LIN {X 0,Y 411.222,Z 293.884,A -85,B 0,C 180,E1 -10421.051,E2 -10421.051} C_VEL
LIN {X 0,Y 411.251,Z 293.88,A -85,B 0,C 180,E1 -10424.131,E2 -10424.131} C_VEL
LIN {X 0,Y 411.3,Z 293.873,A -85,B 0,C 180,E1 -10427.165,E2 -10427.165} C_VEL
LIN {X 0,Y 411.29,Z 293.877,A -85,B 0,C 180,E1 -10430.161,E2 -10430.161} C_VEL
LIN {X 0,Y 411.391,Z 293.865,A -85,B 0,C 180,E1 -10433.132,E2 -10433.132} C_VEL
LIN {X 0,Y 411.304,Z 293.877,A -85,B 0,C 180,E1 -10435.099,E2 -10435.099} C_VEL
LIN {X 0,Y 411.511,Z 293.85,A -85,B 0,C 180,E1 -10438.042,E2 -10438.042} C_VEL
LIN {X 0,Y 411.632,Z 293.838,A -85,B 0,C 180,E1 -10440,E2 -10440} C_VEL
LIN {X 0,Y 411.464,Z 293.859,A -85,B 0,C 180,E1 -10442.937,E2 -10442.937} C_VEL
LIN {X 0,Y 411.433,Z 293.861,A -85,B 0,C 180,E1 -10445.882,E2 -10445.882} C_VEL
LIN {X 0,Y 411.316,Z 293.875,A -85,B 0,C 180,E1 -10448.846,E2 -10448.846} C_VEL
LIN {X 0,Y 411.281,Z 293.88,A -85,B 0,C 180,E1 -10451.833,E2 -10451.833} C_VEL
LIN {X 0,Y 411.256,Z 293.883,A -85,B 0,C 180,E1 -10454.853,E2 -10454.853} C_VEL
LIN {X 0,Y 411.249,Z 293.883,A -85,B 0,C 180,E1 -10457.915,E2 -10457.915} C_VEL
LIN {X 0,Y 411.193,Z 293.89,A -85,B 0,C 180,E1 -10461.034,E2 -10461.034} C_VEL
LIN {X 0,Y 411.217,Z 293.888,A -85,B 0,C 180,E1 -10464.216,E2 -10464.216} C_VEL
LIN {X 0,Y 411.256,Z 293.886,A -85,B 0,C 180,E1 -10467.478,E2 -10467.478} C_VEL
LIN {X 0,Y 411.187,Z 293.897,A -85,B 0,C 180,E1 -10470.848,E2 -10470.848} C_VEL
LIN {X 0,Y 411.203,Z 293.895,A -85,B 0,C 180,E1 -10474.334,E2 -10474.334} C_VEL
LIN {X 0,Y 411.188,Z 293.897,A -85,B 0,C 180,E1 -10477.974,E2 -10477.974} C_VEL
LIN {X 0,Y 411.158,Z 293.897,A -85,B 0,C 180,E1 -10481.228,E2 -10481.228} C_VEL
LIN {X 0,Y 411.22,Z 294.123,A -85,B 0,C 180,E1 -10483.127,E2 -10483.127} C_VEL
LIN {X 0,Y 411.74,Z 297.377,A -85,B 0,C 180,E1 -10485.799,E2 -10485.799} C_VEL
LIN {X 0,Y 412.024,Z 301.04,A -85,B 0,C 180,E1 -10488.635,E2 -10488.635} C_VEL
LIN {X 0,Y 411.836,Z 305.321,A -85,B 0,C 180,E1 -10491.72,E2 -10491.72} C_VEL
LIN {X 0,Y 411.501,Z 310.164,A -85,B 0,C 180,E1 -10495.063,E2 -10495.063} C_VEL
LIN {X 0,Y 411.137,Z 315.732,A -85,B 0,C 180,E1 -10498.727,E2 -10498.727} C_VEL
LIN {X 0,Y 410.779,Z 321.654,A -85,B 0,C 180,E1 -10502.488,E2 -10502.488} C_VEL
LIN {X 0,Y 410.569,Z 325.761,A -85,B 0,C 180,E1 -10505.017,E2 -10505.017} C_VEL
LIN {X 0,Y 412.96,Z 333.703,A -85,B 0,C 180,E1 -10505.349,E2 -10505.349} C_VEL
LIN {X 0,Y 417.044,Z 348.163,A -85,B 0,C 180,E1 -10506.057,E2 -10506.057} C_VEL
LIN {X 0,Y 420.257,Z 362.682,A -85,B 0,C 180,E1 -10506.892,E2 -10506.892} C_VEL
LIN {X 0,Y 419.468,Z 375.628,A -85,B 0,C 180,E1 -10507.594,E2 -10507.594} C_VEL
LIN {X 0,Y 418.211,Z 389.915,A -85,B 0,C 180,E1 -10508.561,E2 -10508.561} C_VEL
LIN {X 0,Y 416.924,Z 402.918,A -85,B 0,C 180,E1 -10509.655,E2 -10509.655} C_VEL
LIN {X 0,Y 415.653,Z 414.924,A -85,B 0,C 180,E1 -10510.877,E2 -10510.877} C_VEL
LIN {X 0,Y 414.497,Z 426.042,A -85,B 0,C 180,E1 -10512.23,E2 -10512.23} C_VEL
LIN {X 0,Y 413.333,Z 436.268,A -85,B 0,C 180,E1 -10513.707,E2 -10513.707} C_VEL
LIN {X 0,Y 412.281,Z 446.263,A -85,B 0,C 180,E1 -10515.437,E2 -10515.437} C_VEL
LIN {X 0,Y 411.345,Z 455.643,A -85,B 0,C 180,E1 -10517.418,E2 -10517.418} C_VEL
LIN {X 0,Y 410.772,Z 462.357,A -85,B 0,C 180,E1 -10519.152,E2 -10519.152} C_VEL
LIN {X 0,Y 410.337,Z 468.557,A -85,B 0,C 180,E1 -10521.132,E2 -10521.132} C_VEL
LIN {X 0,Y 410.082,Z 473.352,A -85,B 0,C 180,E1 -10523.11,E2 -10523.11} C_VEL
LIN {X 0,Y 409.968,Z 476.864,A -85,B 0,C 180,E1 -10525.083,E2 -10525.083} C_VEL
LIN {X 0,Y 409.871,Z 479.174,A -85,B 0,C 180,E1 -10527.051,E2 -10527.051} C_VEL
LIN {X 0,Y 409.915,Z 480.337,A -85,B 0,C 180,E1 -10529.017,E2 -10529.017} C_VEL
LIN {X 0,Y 409.915,Z 480.336,A -85,B 0,C 180,E1 -10530.982,E2 -10530.982} C_VEL
LIN {X 0,Y 409.871,Z 479.168,A -85,B 0,C 180,E1 -10532.948,E2 -10532.948} C_VEL
LIN {X 0,Y 409.973,Z 476.855,A -85,B 0,C 180,E1 -10534.917,E2 -10534.917} C_VEL
LIN {X 0,Y 410.155,Z 473.347,A -85,B 0,C 180,E1 -10536.888,E2 -10536.888} C_VEL
LIN {X 0,Y 410.336,Z 468.551,A -85,B 0,C 180,E1 -10538.867,E2 -10538.867} C_VEL
LIN {X 0,Y 410.77,Z 462.34,A -85,B 0,C 180,E1 -10540.847,E2 -10540.847} C_VEL
LIN {X 0,Y 411.351,Z 455.622,A -85,B 0,C 180,E1 -10542.581,E2 -10542.581} C_VEL
LIN {X 0,Y 412.28,Z 446.241,A -85,B 0,C 180,E1 -10544.562,E2 -10544.562} C_VEL
LIN {X 0,Y 413.305,Z 436.241,A -85,B 0,C 180,E1 -10546.294,E2 -10546.294} C_VEL
LIN {X 0,Y 414.63,Z 424.769,A -85,B 0,C 180,E1 -10547.932,E2 -10547.932} C_VEL
LIN {X 0,Y 415.905,Z 412.674,A -85,B 0,C 180,E1 -10549.367,E2 -10549.367} C_VEL
LIN {X 0,Y 417.181,Z 400.249,A -85,B 0,C 180,E1 -10550.589,E2 -10550.589} C_VEL
LIN {X 0,Y 418.477,Z 386.636,A -85,B 0,C 180,E1 -10551.682,E2 -10551.682} C_VEL
LIN {X 0,Y 419.727,Z 372.535,A -85,B 0,C 180,E1 -10552.585,E2 -10552.585} C_VEL
LIN {X 0,Y 420.235,Z 362.738,A -85,B 0,C 180,E1 -10553.101,E2 -10553.101} C_VEL
LIN {X 0,Y 417.1,Z 348.446,A -85,B 0,C 180,E1 -10553.923,E2 -10553.923} C_VEL
LIN {X 0,Y 412.798,Z 333.269,A -85,B 0,C 180,E1 -10554.663,E2 -10554.663} C_VEL
LIN {X 0,Y 410.566,Z 325.765,A -85,B 0,C 180,E1 -10554.987,E2 -10554.987} C_VEL
LIN {X 0,Y 410.775,Z 321.686,A -85,B 0,C 180,E1 -10557.512,E2 -10557.512} C_VEL
LIN {X 0,Y 411.141,Z 315.788,A -85,B 0,C 180,E1 -10561.274,E2 -10561.274} C_VEL
LIN {X 0,Y 411.505,Z 310.225,A -85,B 0,C 180,E1 -10564.937,E2 -10564.937} C_VEL
LIN {X 0,Y 411.833,Z 305.34,A -85,B 0,C 180,E1 -10568.28,E2 -10568.28} C_VEL
LIN {X 0,Y 412.015,Z 300.592,A -85,B 0,C 180,E1 -10571.7,E2 -10571.7} C_VEL
LIN {X 0,Y 411.705,Z 297.085,A -85,B 0,C 180,E1 -10574.417,E2 -10574.417} C_VEL
LIN {X 0,Y 411.217,Z 294.096,A -85,B 0,C 180,E1 -10576.872,E2 -10576.872} C_VEL
LIN {X 0,Y 411.208,Z 293.892,A -85,B 0,C 180,E1 -10580.271,E2 -10580.271} C_VEL
LIN {X 0,Y 411.186,Z 293.896,A -85,B 0,C 180,E1 -10583.447,E2 -10583.447} C_VEL
LIN {X 0,Y 411.2,Z 293.894,A -85,B 0,C 180,E1 -10586.873,E2 -10586.873} C_VEL
LIN {X 0,Y 411.225,Z 293.891,A -85,B 0,C 180,E1 -10590.644,E2 -10590.644} C_VEL
LIN {X 0,Y 411.23,Z 293.888,A -85,B 0,C 180,E1 -10593.619,E2 -10593.619} C_VEL
LIN {X 0,Y 411.195,Z 293.891,A -85,B 0,C 180,E1 -10596.852,E2 -10596.852} C_VEL
LIN {X 0,Y 411.207,Z 293.89,A -85,B 0,C 180,E1 -10600.05,E2 -10600.05} C_VEL
LIN {X 0,Y 411.255,Z 293.883,A -85,B 0,C 180,E1 -10603.131,E2 -10603.131} C_VEL
LIN {X 0,Y 411.297,Z 293.877,A -85,B 0,C 180,E1 -10606.896,E2 -10606.896} C_VEL
LIN {X 0,Y 411.285,Z 293.878,A -85,B 0,C 180,E1 -10610.161,E2 -10610.161} C_VEL
LIN {X 0,Y 411.386,Z 293.865,A -85,B 0,C 180,E1 -10613.132,E2 -10613.132} C_VEL
LIN {X 0,Y 411.301,Z 293.875,A -85,B 0,C 180,E1 -10615.099,E2 -10615.099} C_VEL
LIN {X 0,Y 411.506,Z 293.848,A -85,B 0,C 180,E1 -10618.043,E2 -10618.043} C_VEL
LIN {X 0,Y 411.629,Z 293.838,A -85,B 0,C 180,E1 -10620,E2 -10620} C_VEL
LIN {X 0,Y 411.46,Z 293.859,A -85,B 0,C 180,E1 -10622.937,E2 -10622.937} C_VEL
LIN {X 0,Y 411.389,Z 293.864,A -85,B 0,C 180,E1 -10626.45,E2 -10626.45} C_VEL
LIN {X 0,Y 411.311,Z 293.873,A -85,B 0,C 180,E1 -10628.846,E2 -10628.846} C_VEL
LIN {X 0,Y 411.276,Z 293.877,A -85,B 0,C 180,E1 -10631.833,E2 -10631.833} C_VEL
LIN {X 0,Y 411.251,Z 293.881,A -85,B 0,C 180,E1 -10634.853,E2 -10634.853} C_VEL
LIN {X 0,Y 411.245,Z 293.882,A -85,B 0,C 180,E1 -10637.916,E2 -10637.916} C_VEL
LIN {X 0,Y 411.189,Z 293.89,A -85,B 0,C 180,E1 -10641.035,E2 -10641.035} C_VEL
LIN {X 0,Y 411.22,Z 293.888,A -85,B 0,C 180,E1 -10644.216,E2 -10644.216} C_VEL
LIN {X 0,Y 411.252,Z 293.884,A -85,B 0,C 180,E1 -10647.478,E2 -10647.478} C_VEL
LIN {X 0,Y 411.183,Z 293.89,A -85,B 0,C 180,E1 -10650.848,E2 -10650.848} C_VEL
LIN {X 0,Y 411.199,Z 293.887,A -85,B 0,C 180,E1 -10654.334,E2 -10654.334} C_VEL
LIN {X 0,Y 411.191,Z 293.892,A -85,B 0,C 180,E1 -10657.974,E2 -10657.974} C_VEL
LIN {X 0,Y 411.178,Z 293.893,A -85,B 0,C 180,E1 -10660.505,E2 -10660.505} C_VEL
LIN {X 0,Y 411.168,Z 293.895,A -85,B 0,C 180,E1 -10663.134,E2 -10663.134} C_VEL
LIN {X 0,Y 411.172,Z 293.896,A -85,B 0,C 180,E1 -10664.491,E2 -10664.491} C_VEL
LIN {X 0,Y 411.298,Z 294.707,A -85,B 0,C 180,E1 -10665.863,E2 -10665.863} C_VEL
LIN {X 0,Y 411.549,Z 297.88,A -85,B 0,C 180,E1 -10668.711,E2 -10668.711} C_VEL
LIN {X 0,Y 411.484,Z 300.347,A -85,B 0,C 180,E1 -10670.807,E2 -10670.807} C_VEL
LIN {X 0,Y 411.247,Z 304.858,A -85,B 0,C 180,E1 -10674.477,E2 -10674.477} C_VEL
LIN {X 0,Y 410.983,Z 309.361,A -85,B 0,C 180,E1 -10677.988,E2 -10677.988} C_VEL
LIN {X 0,Y 410.73,Z 313.896,A -85,B 0,C 180,E1 -10681.374,E2 -10681.374} C_VEL
LIN {X 0,Y 410.532,Z 319.007,A -85,B 0,C 180,E1 -10685.077,E2 -10685.077} C_VEL
LIN {X 0,Y 412.277,Z 324.668,A -85,B 0,C 180,E1 -10685.319,E2 -10685.319} C_VEL
LIN {X 0,Y 416.954,Z 339.922,A -85,B 0,C 180,E1 -10686.073,E2 -10686.073} C_VEL
LIN {X 0,Y 420.328,Z 353.637,A -85,B 0,C 180,E1 -10686.87,E2 -10686.87} C_VEL
LIN {X 0,Y 420.411,Z 357.047,A -85,B 0,C 180,E1 -10687.046,E2 -10687.046} C_VEL
LIN {X 0,Y 419.384,Z 371.28,A -85,B 0,C 180,E1 -10687.85,E2 -10687.85} C_VEL
LIN {X 0,Y 418.122,Z 384.886,A -85,B 0,C 180,E1 -10688.816,E2 -10688.816} C_VEL
LIN {X 0,Y 416.783,Z 398.69,A -85,B 0,C 180,E1 -10690.035,E2 -10690.035} C_VEL
LIN {X 0,Y 415.437,Z 411.499,A -85,B 0,C 180,E1 -10691.422,E2 -10691.422} C_VEL
LIN {X 0,Y 414.159,Z 423.349,A -85,B 0,C 180,E1 -10692.98,E2 -10692.98} C_VEL
LIN {X 0,Y 412.951,Z 434.189,A -85,B 0,C 180,E1 -10694.705,E2 -10694.705} C_VEL
LIN {X 0,Y 411.883,Z 443.751,A -85,B 0,C 180,E1 -10696.556,E2 -10696.556} C_VEL
LIN {X 0,Y 411.341,Z 450.645,A -85,B 0,C 180,E1 -10698.17,E2 -10698.17} C_VEL
LIN {X 0,Y 410.673,Z 457.62,A -85,B 0,C 180,E1 -10700.147,E2 -10700.147} C_VEL
LIN {X 0,Y 410.272,Z 463.102,A -85,B 0,C 180,E1 -10702.124,E2 -10702.124} C_VEL
LIN {X 0,Y 410.06,Z 467.242,A -85,B 0,C 180,E1 -10704.098,E2 -10704.098} C_VEL
LIN {X 0,Y 409.919,Z 470.153,A -85,B 0,C 180,E1 -10706.068,E2 -10706.068} C_VEL
LIN {X 0,Y 409.964,Z 471.904,A -85,B 0,C 180,E1 -10708.036,E2 -10708.036} C_VEL
LIN {X 0,Y 409.904,Z 472.517,A -85,B 0,C 180,E1 -10710,E2 -10710} C_VEL
LIN {X 0,Y 409.965,Z 471.952,A -85,B 0,C 180,E1 -10711.965,E2 -10711.965} C_VEL
LIN {X 0,Y 409.918,Z 470.264,A -85,B 0,C 180,E1 -10713.933,E2 -10713.933} C_VEL
LIN {X 0,Y 410.053,Z 467.413,A -85,B 0,C 180,E1 -10715.903,E2 -10715.903} C_VEL
LIN {X 0,Y 410.169,Z 465.034,A -85,B 0,C 180,E1 -10717.121,E2 -10717.121} C_VEL
LIN {X 0,Y 409.551,Z 463.32,A -85,B 0,C 180,E1 -10717.907,E2 -10717.907} C_VEL
LIN {X 0,Y 406.84,Z 460.256,A -85,B 0,C 180,E1 -10719.179,E2 -10719.179} C_VEL
LIN {X 0,Y 404.299,Z 456.695,A -85,B 0,C 180,E1 -10720.439,E2 -10720.439} C_VEL
LIN {X 0,Y 403.951,Z 454.165,A -85,B 0,C 180,E1 -10721.196,E2 -10721.196} C_VEL
LIN {X 0,Y 404.536,Z 448.082,A -85,B 0,C 180,E1 -10722.798,E2 -10722.798} C_VEL
LIN {X 0,Y 405.494,Z 438.803,A -85,B 0,C 180,E1 -10724.812,E2 -10724.812} C_VEL
LIN {X 0,Y 406.669,Z 428.898,A -85,B 0,C 180,E1 -10726.568,E2 -10726.568} C_VEL
LIN {X 0,Y 408.059,Z 417.47,A -85,B 0,C 180,E1 -10728.24,E2 -10728.24} C_VEL
LIN {X 0,Y 409.4,Z 405.552,A -85,B 0,C 180,E1 -10729.688,E2 -10729.688} C_VEL
LIN {X 0,Y 410.75,Z 393.245,A -85,B 0,C 180,E1 -10730.927,E2 -10730.927} C_VEL
LIN {X 0,Y 412.036,Z 379.795,A -85,B 0,C 180,E1 -10732.04,E2 -10732.04} C_VEL
LIN {X 0,Y 413.285,Z 365.857,A -85,B 0,C 180,E1 -10732.958,E2 -10732.958} C_VEL
LIN {X 0,Y 413.862,Z 355.692,A -85,B 0,C 180,E1 -10733.508,E2 -10733.508} C_VEL
LIN {X 0,Y 410.314,Z 341.226,A -85,B 0,C 180,E1 -10734.391,E2 -10734.391} C_VEL
LIN {X 0,Y 405.961,Z 326.76,A -85,B 0,C 180,E1 -10735.144,E2 -10735.144} C_VEL
LIN {X 0,Y 403.515,Z 319.575,A -85,B 0,C 180,E1 -10735.471,E2 -10735.471} C_VEL
LIN {X 0,Y 403.469,Z 319.059,A -85,B 0,C 180,E1 -10735.524,E2 -10735.524} C_VEL
LIN {X 0,Y 403.738,Z 314.147,A -85,B 0,C 180,E1 -10739.17,E2 -10739.17} C_VEL
LIN {X 0,Y 403.985,Z 309.636,A -85,B 0,C 180,E1 -10742.636,E2 -10742.636} C_VEL
LIN {X 0,Y 404.206,Z 306.384,A -85,B 0,C 180,E1 -10745.195,E2 -10745.195} C_VEL
LIN {X 0,Y 404.409,Z 302.079,A -85,B 0,C 180,E1 -10748.728,E2 -10748.728} C_VEL
LIN {X 0,Y 404.552,Z 299.055,A -85,B 0,C 180,E1 -10751.311,E2 -10751.311} C_VEL
LIN {X 0,Y 404.348,Z 296.014,A -85,B 0,C 180,E1 -10754.046,E2 -10754.046} C_VEL
LIN {X 0,Y 404.15,Z 294.772,A -85,B 0,C 180,E1 -10755.477,E2 -10755.477} C_VEL
LIN {X 0,Y 404.118,Z 294.773,A -85,B 0,C 180,E1 -10758.635,E2 -10758.635} C_VEL
LIN {X 0,Y 404.154,Z 294.769,A -85,B 0,C 180,E1 -10761.492,E2 -10761.492} C_VEL
LIN {X 0,Y 404.183,Z 294.768,A -85,B 0,C 180,E1 -10764.984,E2 -10764.984} C_VEL
LIN {X 0,Y 404.14,Z 294.77,A -85,B 0,C 180,E1 -10768.553,E2 -10768.553} C_VEL
LIN {X 0,Y 404.155,Z 294.769,A -85,B 0,C 180,E1 -10770.863,E2 -10770.863} C_VEL
LIN {X 0,Y 404.148,Z 294.77,A -85,B 0,C 180,E1 -10774.231,E2 -10774.231} C_VEL
LIN {X 0,Y 404.165,Z 294.764,A -85,B 0,C 180,E1 -10777.508,E2 -10777.508} C_VEL
LIN {X 0,Y 404.163,Z 294.763,A -85,B 0,C 180,E1 -10780.707,E2 -10780.707} C_VEL
LIN {X 0,Y 404.218,Z 294.756,A -85,B 0,C 180,E1 -10783.848,E2 -10783.848} C_VEL
LIN {X 0,Y 404.28,Z 294.747,A -85,B 0,C 180,E1 -10786.939,E2 -10786.939} C_VEL
LIN {X 0,Y 404.255,Z 294.754,A -85,B 0,C 180,E1 -10789.988,E2 -10789.988} C_VEL
LIN {X 0,Y 404.341,Z 294.743,A -85,B 0,C 180,E1 -10793.011,E2 -10793.011} C_VEL
LIN {X 0,Y 404.274,Z 294.752,A -85,B 0,C 180,E1 -10795.013,E2 -10795.013} C_VEL
LIN {X 0,Y 404.48,Z 294.726,A -85,B 0,C 180,E1 -10798.008,E2 -10798.008} C_VEL
LIN {X 0,Y 404.601,Z 294.713,A -85,B 0,C 180,E1 -10800,E2 -10800} C_VEL
LIN {X 0,Y 404.421,Z 294.736,A -85,B 0,C 180,E1 -10802.988,E2 -10802.988} C_VEL
LIN {X 0,Y 404.381,Z 294.74,A -85,B 0,C 180,E1 -10805.985,E2 -10805.985} C_VEL
LIN {X 0,Y 404.263,Z 294.755,A -85,B 0,C 180,E1 -10809.002,E2 -10809.002} C_VEL
LIN {X 0,Y 404.253,Z 294.757,A -85,B 0,C 180,E1 -10812.041,E2 -10812.041} C_VEL
LIN {X 0,Y 404.202,Z 294.763,A -85,B 0,C 180,E1 -10815.118,E2 -10815.118} C_VEL
LIN {X 0,Y 404.207,Z 294.762,A -85,B 0,C 180,E1 -10818.238,E2 -10818.238} C_VEL
LIN {X 0,Y 404.135,Z 294.772,A -85,B 0,C 180,E1 -10821.419,E2 -10821.419} C_VEL
LIN {X 0,Y 404.171,Z 294.767,A -85,B 0,C 180,E1 -10824.666,E2 -10824.666} C_VEL
LIN {X 0,Y 404.192,Z 294.765,A -85,B 0,C 180,E1 -10828,E2 -10828} C_VEL
LIN {X 0,Y 404.136,Z 294.773,A -85,B 0,C 180,E1 -10831.558,E2 -10831.558} C_VEL
LIN {X 0,Y 404.182,Z 294.771,A -85,B 0,C 180,E1 -10835.016,E2 -10835.016} C_VEL
LIN {X 0,Y 404.146,Z 294.773,A -85,B 0,C 180,E1 -10838.758,E2 -10838.758} C_VEL
LIN {X 0,Y 404.117,Z 294.775,A -85,B 0,C 180,E1 -10841.599,E2 -10841.599} C_VEL
LIN {X 0,Y 404.159,Z 294.854,A -85,B 0,C 180,E1 -10842.701,E2 -10842.701} C_VEL
LIN {X 0,Y 404.687,Z 298.05,A -85,B 0,C 180,E1 -10845.4,E2 -10845.4} C_VEL
LIN {X 0,Y 405.009,Z 301.655,A -85,B 0,C 180,E1 -10848.259,E2 -10848.259} C_VEL
LIN {X 0,Y 404.821,Z 305.87,A -85,B 0,C 180,E1 -10851.373,E2 -10851.373} C_VEL
LIN {X 0,Y 404.471,Z 311.053,A -85,B 0,C 180,E1 -10855.012,E2 -10855.012} C_VEL
LIN {X 0,Y 404.112,Z 316.324,A -85,B 0,C 180,E1 -10858.551,E2 -10858.551} C_VEL
LIN {X 0,Y 403.755,Z 321.601,A -85,B 0,C 180,E1 -10861.967,E2 -10861.967} C_VEL
LIN {X 0,Y 403.516,Z 325.685,A -85,B 0,C 180,E1 -10864.549,E2 -10864.549} C_VEL
LIN {X 0,Y 405.401,Z 331.748,A -85,B 0,C 180,E1 -10864.815,E2 -10864.815} C_VEL
LIN {X 0,Y 409.888,Z 347.21,A -85,B 0,C 180,E1 -10865.58,E2 -10865.58} C_VEL
LIN {X 0,Y 413.149,Z 361.479,A -85,B 0,C 180,E1 -10866.413,E2 -10866.413} C_VEL
LIN {X 0,Y 413.665,Z 364.983,A -85,B 0,C 180,E1 -10866.623,E2 -10866.623} C_VEL
LIN {X 0,Y 412.55,Z 379.541,A -85,B 0,C 180,E1 -10867.462,E2 -10867.462} C_VEL
LIN {X 0,Y 411.285,Z 393.014,A -85,B 0,C 180,E1 -10868.445,E2 -10868.445} C_VEL
LIN {X 0,Y 409.959,Z 405.437,A -85,B 0,C 180,E1 -10869.556,E2 -10869.556} C_VEL
LIN {X 0,Y 408.552,Z 418.07,A -85,B 0,C 180,E1 -10870.923,E2 -10870.923} C_VEL
LIN {X 0,Y 407.269,Z 429.545,A -85,B 0,C 180,E1 -10872.423,E2 -10872.423} C_VEL
LIN {X 0,Y 406.119,Z 439.202,A -85,B 0,C 180,E1 -10873.926,E2 -10873.926} C_VEL
LIN {X 0,Y 405.046,Z 448.685,A -85,B 0,C 180,E1 -10875.685,E2 -10875.685} C_VEL
LIN {X 0,Y 404.255,Z 456.585,A -85,B 0,C 180,E1 -10877.449,E2 -10877.449} C_VEL
LIN {X 0,Y 403.772,Z 462.289,A -85,B 0,C 180,E1 -10878.962,E2 -10878.962} C_VEL
LIN {X 0,Y 403.282,Z 468.489,A -85,B 0,C 180,E1 -10880.976,E2 -10880.976} C_VEL
LIN {X 0,Y 403.003,Z 473.283,A -85,B 0,C 180,E1 -10882.988,E2 -10882.988} C_VEL
LIN {X 0,Y 402.881,Z 476.796,A -85,B 0,C 180,E1 -10884.996,E2 -10884.996} C_VEL
LIN {X 0,Y 402.773,Z 479.105,A -85,B 0,C 180,E1 -10886.999,E2 -10886.999} C_VEL
LIN {X 0,Y 402.842,Z 480.268,A -85,B 0,C 180,E1 -10889,E2 -10889} C_VEL
LIN {X 0,Y 402.842,Z 480.267,A -85,B 0,C 180,E1 -10890.999,E2 -10890.999} C_VEL
LIN {X 0,Y 402.773,Z 479.098,A -85,B 0,C 180,E1 -10893,E2 -10893} C_VEL
LIN {X 0,Y 402.888,Z 476.786,A -85,B 0,C 180,E1 -10895.003,E2 -10895.003} C_VEL
LIN {X 0,Y 403.065,Z 473.277,A -85,B 0,C 180,E1 -10897.01,E2 -10897.01} C_VEL
LIN {X 0,Y 403.282,Z 468.481,A -85,B 0,C 180,E1 -10899.023,E2 -10899.023} C_VEL
LIN {X 0,Y 403.769,Z 462.27,A -85,B 0,C 180,E1 -10901.038,E2 -10901.038} C_VEL
LIN {X 0,Y 404.374,Z 455.551,A -85,B 0,C 180,E1 -10902.802,E2 -10902.802} C_VEL
LIN {X 0,Y 405.179,Z 447.427,A -85,B 0,C 180,E1 -10904.566,E2 -10904.566} C_VEL
LIN {X 0,Y 406.27,Z 437.686,A -85,B 0,C 180,E1 -10906.326,E2 -10906.326} C_VEL
LIN {X 0,Y 407.496,Z 427.725,A -85,B 0,C 180,E1 -10907.825,E2 -10907.825} C_VEL
LIN {X 0,Y 408.774,Z 415.891,A -85,B 0,C 180,E1 -10909.326,E2 -10909.326} C_VEL
LIN {X 0,Y 410.072,Z 404.097,A -85,B 0,C 180,E1 -10910.568,E2 -10910.568} C_VEL
LIN {X 0,Y 411.395,Z 391.358,A -85,B 0,C 180,E1 -10911.68,E2 -10911.68} C_VEL
LIN {X 0,Y 412.751,Z 377.458,A -85,B 0,C 180,E1 -10912.658,E2 -10912.658} C_VEL
LIN {X 0,Y 413.601,Z 363.995,A -85,B 0,C 180,E1 -10913.425,E2 -10913.425} C_VEL
LIN {X 0,Y 410.533,Z 349.912,A -85,B 0,C 180,E1 -10914.273,E2 -10914.273} C_VEL
LIN {X 0,Y 406.175,Z 334.223,A -85,B 0,C 180,E1 -10915.069,E2 -10915.069} C_VEL
LIN {X 0,Y 403.598,Z 326.284,A -85,B 0,C 180,E1 -10915.419,E2 -10915.419} C_VEL
LIN {X 0,Y 403.513,Z 325.695,A -85,B 0,C 180,E1 -10915.45,E2 -10915.45} C_VEL
LIN {X 0,Y 403.751,Z 321.629,A -85,B 0,C 180,E1 -10918.032,E2 -10918.032} C_VEL
LIN {X 0,Y 404.114,Z 316.217,A -85,B 0,C 180,E1 -10921.552,E2 -10921.552} C_VEL
LIN {X 0,Y 404.508,Z 310.713,A -85,B 0,C 180,E1 -10925.256,E2 -10925.256} C_VEL
LIN {X 0,Y 404.822,Z 305.814,A -85,B 0,C 180,E1 -10928.68,E2 -10928.68} C_VEL
LIN {X 0,Y 405.007,Z 301.658,A -85,B 0,C 180,E1 -10931.74,E2 -10931.74} C_VEL
LIN {X 0,Y 404.687,Z 298.03,A -85,B 0,C 180,E1 -10934.6,E2 -10934.6} C_VEL
LIN {X 0,Y 404.159,Z 294.826,A -85,B 0,C 180,E1 -10937.299,E2 -10937.299} C_VEL
LIN {X 0,Y 404.163,Z 294.769,A -85,B 0,C 180,E1 -10939.955,E2 -10939.955} C_VEL
LIN {X 0,Y 404.129,Z 294.774,A -85,B 0,C 180,E1 -10943.125,E2 -10943.125} C_VEL
LIN {X 0,Y 404.138,Z 294.775,A -85,B 0,C 180,E1 -10946.187,E2 -10946.187} C_VEL
LIN {X 0,Y 404.138,Z 294.774,A -85,B 0,C 180,E1 -10949.714,E2 -10949.714} C_VEL
LIN {X 0,Y 404.188,Z 294.764,A -85,B 0,C 180,E1 -10953.122,E2 -10953.122} C_VEL
LIN {X 0,Y 404.17,Z 294.767,A -85,B 0,C 180,E1 -10955.334,E2 -10955.334} C_VEL
LIN {X 0,Y 404.131,Z 294.771,A -85,B 0,C 180,E1 -10958.58,E2 -10958.58} C_VEL
LIN {X 0,Y 404.202,Z 294.762,A -85,B 0,C 180,E1 -10961.762,E2 -10961.762} C_VEL
LIN {X 0,Y 404.197,Z 294.761,A -85,B 0,C 180,E1 -10964.882,E2 -10964.882} C_VEL
LIN {X 0,Y 404.249,Z 294.755,A -85,B 0,C 180,E1 -10967.958,E2 -10967.958} C_VEL
LIN {X 0,Y 404.258,Z 294.753,A -85,B 0,C 180,E1 -10970.998,E2 -10970.998} C_VEL
LIN {X 0,Y 404.376,Z 294.738,A -85,B 0,C 180,E1 -10974.014,E2 -10974.014} C_VEL
LIN {X 0,Y 404.475,Z 294.723,A -85,B 0,C 180,E1 -10978.009,E2 -10978.009} C_VEL
LIN {X 0,Y 404.598,Z 294.714,A -85,B 0,C 180,E1 -10980,E2 -10980} C_VEL
LIN {X 0,Y 404.417,Z 294.737,A -85,B 0,C 180,E1 -10982.989,E2 -10982.989} C_VEL
LIN {X 0,Y 404.342,Z 294.742,A -85,B 0,C 180,E1 -10986.443,E2 -10986.443} C_VEL
LIN {X 0,Y 404.258,Z 294.753,A -85,B 0,C 180,E1 -10989.002,E2 -10989.002} C_VEL
LIN {X 0,Y 404.249,Z 294.754,A -85,B 0,C 180,E1 -10992.042,E2 -10992.042} C_VEL
LIN {X 0,Y 404.198,Z 294.761,A -85,B 0,C 180,E1 -10995.118,E2 -10995.118} C_VEL
LIN {X 0,Y 404.203,Z 294.761,A -85,B 0,C 180,E1 -10998.239,E2 -10998.239} C_VEL
LIN {X 0,Y 404.152,Z 294.77,A -85,B 0,C 180,E1 -11001.419,E2 -11001.419} C_VEL
LIN {X 0,Y 404.171,Z 294.766,A -85,B 0,C 180,E1 -11004.666,E2 -11004.666} C_VEL
LIN {X 0,Y 404.188,Z 294.76,A -85,B 0,C 180,E1 -11008,E2 -11008} C_VEL
LIN {X 0,Y 404.133,Z 294.766,A -85,B 0,C 180,E1 -11011.559,E2 -11011.559} C_VEL
LIN {X 0,Y 404.178,Z 294.763,A -85,B 0,C 180,E1 -11015.017,E2 -11015.017} C_VEL
LIN {X 0,Y 404.152,Z 294.768,A -85,B 0,C 180,E1 -11018.757,E2 -11018.757} C_VEL
LIN {X 0,Y 404.119,Z 294.775,A -85,B 0,C 180,E1 -11021.601,E2 -11021.601} C_VEL
LIN {X 0,Y 404.141,Z 294.772,A -85,B 0,C 180,E1 -11024.523,E2 -11024.523} C_VEL
LIN {X 0,Y 404.302,Z 295.896,A -85,B 0,C 180,E1 -11025.949,E2 -11025.949} C_VEL
LIN {X 0,Y 404.544,Z 298.898,A -85,B 0,C 180,E1 -11028.689,E2 -11028.689} C_VEL
LIN {X 0,Y 404.388,Z 302.118,A -85,B 0,C 180,E1 -11031.451,E2 -11031.451} C_VEL
LIN {X 0,Y 404.195,Z 306.409,A -85,B 0,C 180,E1 -11034.986,E2 -11034.986} C_VEL
LIN {X 0,Y 403.896,Z 310.936,A -85,B 0,C 180,E1 -11038.533,E2 -11038.533} C_VEL
LIN {X 0,Y 403.621,Z 315.472,A -85,B 0,C 180,E1 -11041.958,E2 -11041.958} C_VEL
LIN {X 0,Y 403.497,Z 319.079,A -85,B 0,C 180,E1 -11044.609,E2 -11044.609} C_VEL
LIN {X 0,Y 405.399,Z 325.071,A -85,B 0,C 180,E1 -11044.879,E2 -11044.879} C_VEL
LIN {X 0,Y 410.131,Z 340.418,A -85,B 0,C 180,E1 -11045.665,E2 -11045.665} C_VEL
LIN {X 0,Y 413.695,Z 355.042,A -85,B 0,C 180,E1 -11046.545,E2 -11046.545} C_VEL
LIN {X 0,Y 413.873,Z 357.231,A -85,B 0,C 180,E1 -11046.668,E2 -11046.668} C_VEL
LIN {X 0,Y 412.822,Z 371.356,A -85,B 0,C 180,E1 -11047.478,E2 -11047.478} C_VEL
LIN {X 0,Y 411.501,Z 384.961,A -85,B 0,C 180,E1 -11048.458,E2 -11048.458} C_VEL
LIN {X 0,Y 410.098,Z 398.764,A -85,B 0,C 180,E1 -11049.695,E2 -11049.695} C_VEL
LIN {X 0,Y 408.755,Z 410.893,A -85,B 0,C 180,E1 -11051.024,E2 -11051.024} C_VEL
LIN {X 0,Y 407.502,Z 421.648,A -85,B 0,C 180,E1 -11052.434,E2 -11052.434} C_VEL
LIN {X 0,Y 406.376,Z 431.324,A -85,B 0,C 180,E1 -11053.937,E2 -11053.937} C_VEL
LIN {X 0,Y 405.28,Z 440.81,A -85,B 0,C 180,E1 -11055.694,E2 -11055.694} C_VEL
LIN {X 0,Y 404.533,Z 448.707,A -85,B 0,C 180,E1 -11057.458,E2 -11057.458} C_VEL
LIN {X 0,Y 403.752,Z 456.083,A -85,B 0,C 180,E1 -11059.469,E2 -11059.469} C_VEL
LIN {X 0,Y 403.319,Z 461.936,A -85,B 0,C 180,E1 -11061.483,E2 -11061.483} C_VEL
LIN {X 0,Y 403.075,Z 465.402,A -85,B 0,C 180,E1 -11062.99,E2 -11062.99} C_VEL
LIN {X 0,Y 402.926,Z 468.916,A -85,B 0,C 180,E1 -11064.997,E2 -11064.997} C_VEL
LIN {X 0,Y 402.819,Z 471.24,A -85,B 0,C 180,E1 -11067,E2 -11067} C_VEL
LIN {X 0,Y 402.845,Z 472.427,A -85,B 0,C 180,E1 -11069.001,E2 -11069.001} C_VEL
LIN {X 0,Y 402.846,Z 472.443,A -85,B 0,C 180,E1 -11071,E2 -11071} C_VEL
LIN {X 0,Y 402.819,Z 471.319,A -85,B 0,C 180,E1 -11073.001,E2 -11073.001} C_VEL
LIN {X 0,Y 402.921,Z 469.056,A -85,B 0,C 180,E1 -11075.004,E2 -11075.004} C_VEL
LIN {X 0,Y 403.087,Z 465.314,A -85,B 0,C 180,E1 -11077.146,E2 -11077.146} C_VEL
LIN {X 0,Y 403.403,Z 460.869,A -85,B 0,C 180,E1 -11079.021,E2 -11079.021} C_VEL
LIN {X 0,Y 403.874,Z 454.741,A -85,B 0,C 180,E1 -11081.036,E2 -11081.036} C_VEL
LIN {X 0,Y 403.951,Z 454.165,A -85,B 0,C 180,E1 -11081.196,E2 -11081.196} C_VEL
LIN {X 0,Y 403.61,Z 451.567,A -85,B 0,C 180,E1 -11081.94,E2 -11081.94} C_VEL
LIN {X 0,Y 401.196,Z 447.104,A -85,B 0,C 180,E1 -11083.153,E2 -11083.153} C_VEL
LIN {X 0,Y 398.835,Z 442.25,A -85,B 0,C 180,E1 -11084.351,E2 -11084.351} C_VEL
LIN {X 0,Y 398.598,Z 438.929,A -85,B 0,C 180,E1 -11085.062,E2 -11085.062} C_VEL
LIN {X 0,Y 399.813,Z 428.965,A -85,B 0,C 180,E1 -11086.861,E2 -11086.861} C_VEL
LIN {X 0,Y 401.261,Z 417.682,A -85,B 0,C 180,E1 -11088.54,E2 -11088.54} C_VEL
LIN {X 0,Y 402.664,Z 405.617,A -85,B 0,C 180,E1 -11090.031,E2 -11090.031} C_VEL
LIN {X 0,Y 404.086,Z 393.309,A -85,B 0,C 180,E1 -11091.289,E2 -11091.289} C_VEL
LIN {X 0,Y 405.452,Z 379.858,A -85,B 0,C 180,E1 -11092.417,E2 -11092.417} C_VEL
LIN {X 0,Y 406.799,Z 365.45,A -85,B 0,C 180,E1 -11093.377,E2 -11093.377} C_VEL
LIN {X 0,Y 407.262,Z 356.956,A -85,B 0,C 180,E1 -11093.85,E2 -11093.85} C_VEL
LIN {X 0,Y 403.737,Z 342.537,A -85,B 0,C 180,E1 -11094.768,E2 -11094.768} C_VEL
LIN {X 0,Y 399.097,Z 327.214,A -85,B 0,C 180,E1 -11095.598,E2 -11095.598} C_VEL
LIN {X 0,Y 396.531,Z 319.909,A -85,B 0,C 180,E1 -11095.947,E2 -11095.947} C_VEL
LIN {X 0,Y 396.422,Z 319.168,A -85,B 0,C 180,E1 -11095.977,E2 -11095.977} C_VEL
LIN {X 0,Y 396.626,Z 315.722,A -85,B 0,C 180,E1 -11098.583,E2 -11098.583} C_VEL
LIN {X 0,Y 396.885,Z 311.21,A -85,B 0,C 180,E1 -11102.089,E2 -11102.089} C_VEL
LIN {X 0,Y 397.191,Z 306.673,A -85,B 0,C 180,E1 -11105.726,E2 -11105.726} C_VEL
LIN {X 0,Y 397.426,Z 302.142,A -85,B 0,C 180,E1 -11109.54,E2 -11109.54} C_VEL
LIN {X 0,Y 397.474,Z 299.096,A -85,B 0,C 180,E1 -11112.214,E2 -11112.214} C_VEL
LIN {X 0,Y 397.17,Z 296.058,A -85,B 0,C 180,E1 -11115.056,E2 -11115.056} C_VEL
LIN {X 0,Y 397.102,Z 295.649,A -85,B 0,C 180,E1 -11116.521,E2 -11116.521} C_VEL
LIN {X 0,Y 397.113,Z 295.648,A -85,B 0,C 180,E1 -11120.423,E2 -11120.423} C_VEL
LIN {X 0,Y 397.106,Z 295.647,A -85,B 0,C 180,E1 -11124.265,E2 -11124.265} C_VEL
LIN {X 0,Y 397.113,Z 295.647,A -85,B 0,C 180,E1 -11126.727,E2 -11126.727} C_VEL
LIN {X 0,Y 397.116,Z 295.644,A -85,B 0,C 180,E1 -11130.295,E2 -11130.295} C_VEL
LIN {X 0,Y 397.093,Z 295.646,A -85,B 0,C 180,E1 -11133.739,E2 -11133.739} C_VEL
LIN {X 0,Y 397.101,Z 295.647,A -85,B 0,C 180,E1 -11137.085,E2 -11137.085} C_VEL
LIN {X 0,Y 397.146,Z 295.639,A -85,B 0,C 180,E1 -11140.353,E2 -11140.353} C_VEL
LIN {X 0,Y 397.164,Z 295.635,A -85,B 0,C 180,E1 -11143.553,E2 -11143.553} C_VEL
LIN {X 0,Y 397.226,Z 295.626,A -85,B 0,C 180,E1 -11146.703,E2 -11146.703} C_VEL
LIN {X 0,Y 397.215,Z 295.631,A -85,B 0,C 180,E1 -11149.809,E2 -11149.809} C_VEL
LIN {X 0,Y 397.293,Z 295.621,A -85,B 0,C 180,E1 -11152.887,E2 -11152.887} C_VEL
LIN {X 0,Y 397.244,Z 295.628,A -85,B 0,C 180,E1 -11154.925,E2 -11154.925} C_VEL
LIN {X 0,Y 397.449,Z 295.602,A -85,B 0,C 180,E1 -11157.973,E2 -11157.973} C_VEL
LIN {X 0,Y 397.571,Z 295.589,A -85,B 0,C 180,E1 -11160,E2 -11160} C_VEL
LIN {X 0,Y 397.379,Z 295.613,A -85,B 0,C 180,E1 -11163.041,E2 -11163.041} C_VEL
LIN {X 0,Y 397.331,Z 295.62,A -85,B 0,C 180,E1 -11166.092,E2 -11166.092} C_VEL
LIN {X 0,Y 397.233,Z 295.631,A -85,B 0,C 180,E1 -11169.162,E2 -11169.162} C_VEL
LIN {X 0,Y 397.216,Z 295.634,A -85,B 0,C 180,E1 -11172.258,E2 -11172.258} C_VEL
LIN {X 0,Y 397.176,Z 295.639,A -85,B 0,C 180,E1 -11175.392,E2 -11175.392} C_VEL
LIN {X 0,Y 397.159,Z 295.64,A -85,B 0,C 180,E1 -11178.573,E2 -11178.573} C_VEL
LIN {X 0,Y 397.093,Z 295.647,A -85,B 0,C 180,E1 -11181.819,E2 -11181.819} C_VEL
LIN {X 0,Y 397.15,Z 295.639,A -85,B 0,C 180,E1 -11185.512,E2 -11185.512} C_VEL
LIN {X 0,Y 397.119,Z 295.646,A -85,B 0,C 180,E1 -11188.544,E2 -11188.544} C_VEL
LIN {X 0,Y 397.076,Z 295.656,A -85,B 0,C 180,E1 -11192.072,E2 -11192.072} C_VEL
LIN {X 0,Y 397.117,Z 295.651,A -85,B 0,C 180,E1 -11195.503,E2 -11195.503} C_VEL
LIN {X 0,Y 397.122,Z 295.648,A -85,B 0,C 180,E1 -11198.86,E2 -11198.86} C_VEL
LIN {X 0,Y 397.076,Z 295.651,A -85,B 0,C 180,E1 -11202.266,E2 -11202.266} C_VEL
LIN {X 0,Y 397.624,Z 298.758,A -85,B 0,C 180,E1 -11205.009,E2 -11205.009} C_VEL
LIN {X 0,Y 397.954,Z 302.291,A -85,B 0,C 180,E1 -11207.879,E2 -11207.879} C_VEL
LIN {X 0,Y 397.838,Z 305.733,A -85,B 0,C 180,E1 -11210.509,E2 -11210.509} C_VEL
LIN {X 0,Y 397.612,Z 309.24,A -85,B 0,C 180,E1 -11213.061,E2 -11213.061} C_VEL
LIN {X 0,Y 397.273,Z 313.794,A -85,B 0,C 180,E1 -11216.249,E2 -11216.249} C_VEL
LIN {X 0,Y 396.977,Z 318.011,A -85,B 0,C 180,E1 -11219.109,E2 -11219.109} C_VEL
LIN {X 0,Y 396.661,Z 323.287,A -85,B 0,C 180,E1 -11222.57,E2 -11222.57} C_VEL
LIN {X 0,Y 396.483,Z 325.625,A -85,B 0,C 180,E1 -11224.067,E2 -11224.067} C_VEL
LIN {X 0,Y 398.298,Z 331.51,A -85,B 0,C 180,E1 -11224.329,E2 -11224.329} C_VEL
LIN {X 0,Y 402.861,Z 346.855,A -85,B 0,C 180,E1 -11225.114,E2 -11225.114} C_VEL
LIN {X 0,Y 406.05,Z 360.43,A -85,B 0,C 180,E1 -11225.924,E2 -11225.924} C_VEL
LIN {X 0,Y 407.052,Z 366.443,A -85,B 0,C 180,E1 -11226.308,E2 -11226.308} C_VEL
LIN {X 0,Y 405.969,Z 379.759,A -85,B 0,C 180,E1 -11227.096,E2 -11227.096} C_VEL
LIN {X 0,Y 404.654,Z 392.949,A -85,B 0,C 180,E1 -11228.074,E2 -11228.074} C_VEL
LIN {X 0,Y 403.274,Z 405.371,A -85,B 0,C 180,E1 -11229.201,E2 -11229.201} C_VEL
LIN {X 0,Y 401.792,Z 418.003,A -85,B 0,C 180,E1 -11230.589,E2 -11230.589} C_VEL
LIN {X 0,Y 400.457,Z 429.478,A -85,B 0,C 180,E1 -11232.114,E2 -11232.114} C_VEL
LIN {X 0,Y 399.234,Z 439.134,A -85,B 0,C 180,E1 -11233.641,E2 -11233.641} C_VEL
LIN {X 0,Y 398.114,Z 448.617,A -85,B 0,C 180,E1 -11235.43,E2 -11235.43} C_VEL
LIN {X 0,Y 397.271,Z 456.516,A -85,B 0,C 180,E1 -11237.224,E2 -11237.224} C_VEL
LIN {X 0,Y 396.773,Z 462.22,A -85,B 0,C 180,E1 -11238.764,E2 -11238.764} C_VEL
LIN {X 0,Y 396.239,Z 468.42,A -85,B 0,C 180,E1 -11240.814,E2 -11240.814} C_VEL
LIN {X 0,Y 395.927,Z 473.215,A -85,B 0,C 180,E1 -11242.862,E2 -11242.862} C_VEL
LIN {X 0,Y 395.78,Z 476.727,A -85,B 0,C 180,E1 -11244.906,E2 -11244.906} C_VEL
LIN {X 0,Y 395.679,Z 479.036,A -85,B 0,C 180,E1 -11246.945,E2 -11246.945} C_VEL
LIN {X 0,Y 395.753,Z 480.199,A -85,B 0,C 180,E1 -11248.982,E2 -11248.982} C_VEL
LIN {X 0,Y 395.753,Z 480.198,A -85,B 0,C 180,E1 -11251.017,E2 -11251.017} C_VEL
LIN {X 0,Y 395.679,Z 479.029,A -85,B 0,C 180,E1 -11253.054,E2 -11253.054} C_VEL
LIN {X 0,Y 395.788,Z 476.716,A -85,B 0,C 180,E1 -11255.093,E2 -11255.093} C_VEL
LIN {X 0,Y 395.987,Z 473.207,A -85,B 0,C 180,E1 -11257.136,E2 -11257.136} C_VEL
LIN {X 0,Y 396.238,Z 468.411,A -85,B 0,C 180,E1 -11259.185,E2 -11259.185} C_VEL
LIN {X 0,Y 396.769,Z 462.199,A -85,B 0,C 180,E1 -11261.235,E2 -11261.235} C_VEL
LIN {X 0,Y 397.497,Z 454.397,A -85,B 0,C 180,E1 -11263.288,E2 -11263.288} C_VEL
LIN {X 0,Y 398.415,Z 446.098,A -85,B 0,C 180,E1 -11265.081,E2 -11265.081} C_VEL
LIN {X 0,Y 399.581,Z 436.097,A -85,B 0,C 180,E1 -11266.87,E2 -11266.87} C_VEL
LIN {X 0,Y 400.88,Z 425.868,A -85,B 0,C 180,E1 -11268.394,E2 -11268.394} C_VEL
LIN {X 0,Y 402.325,Z 413.677,A -85,B 0,C 180,E1 -11269.915,E2 -11269.915} C_VEL
LIN {X 0,Y 403.713,Z 401.438,A -85,B 0,C 180,E1 -11271.175,E2 -11271.175} C_VEL
LIN {X 0,Y 405.111,Z 388.116,A -85,B 0,C 180,E1 -11272.302,E2 -11272.302} C_VEL
LIN {X 0,Y 406.431,Z 374.412,A -85,B 0,C 180,E1 -11273.232,E2 -11273.232} C_VEL
LIN {X 0,Y 406.962,Z 365.354,A -85,B 0,C 180,E1 -11273.755,E2 -11273.755} C_VEL
LIN {X 0,Y 403.932,Z 351.289,A -85,B 0,C 180,E1 -11274.633,E2 -11274.633} C_VEL
LIN {X 0,Y 399.91,Z 336.511,A -85,B 0,C 180,E1 -11275.421,E2 -11275.421} C_VEL
LIN {X 0,Y 396.551,Z 326.233,A -85,B 0,C 180,E1 -11275.903,E2 -11275.903} C_VEL
LIN {X 0,Y 396.5,Z 325.588,A -85,B 0,C 180,E1 -11275.961,E2 -11275.961} C_VEL
LIN {X 0,Y 396.729,Z 321.553,A -85,B 0,C 180,E1 -11278.574,E2 -11278.574} C_VEL
LIN {X 0,Y 397.084,Z 316.306,A -85,B 0,C 180,E1 -11282.07,E2 -11282.07} C_VEL
LIN {X 0,Y 397.49,Z 311.211,A -85,B 0,C 180,E1 -11285.578,E2 -11285.578} C_VEL
LIN {X 0,Y 397.803,Z 306.453,A -85,B 0,C 180,E1 -11288.982,E2 -11288.982} C_VEL
LIN {X 0,Y 397.953,Z 304.008,A -85,B 0,C 180,E1 -11290.8,E2 -11290.8} C_VEL
LIN {X 0,Y 397.809,Z 300.445,A -85,B 0,C 180,E1 -11293.586,E2 -11293.586} C_VEL
LIN {X 0,Y 397.327,Z 296.989,A -85,B 0,C 180,E1 -11296.485,E2 -11296.485} C_VEL
LIN {X 0,Y 397.076,Z 295.653,A -85,B 0,C 180,E1 -11297.734,E2 -11297.734} C_VEL
LIN {X 0,Y 397.124,Z 295.644,A -85,B 0,C 180,E1 -11301.138,E2 -11301.138} C_VEL
LIN {X 0,Y 397.112,Z 295.649,A -85,B 0,C 180,E1 -11304.496,E2 -11304.496} C_VEL
LIN {X 0,Y 397.072,Z 295.656,A -85,B 0,C 180,E1 -11307.928,E2 -11307.928} C_VEL
LIN {X 0,Y 397.114,Z 295.647,A -85,B 0,C 180,E1 -11311.456,E2 -11311.456} C_VEL
LIN {X 0,Y 397.145,Z 295.64,A -85,B 0,C 180,E1 -11314.487,E2 -11314.487} C_VEL
LIN {X 0,Y 397.102,Z 295.648,A -85,B 0,C 180,E1 -11317.085,E2 -11317.085} C_VEL
LIN {X 0,Y 397.14,Z 295.641,A -85,B 0,C 180,E1 -11320.353,E2 -11320.353} C_VEL
LIN {X 0,Y 397.158,Z 295.639,A -85,B 0,C 180,E1 -11323.553,E2 -11323.553} C_VEL
LIN {X 0,Y 397.221,Z 295.631,A -85,B 0,C 180,E1 -11326.703,E2 -11326.703} C_VEL
LIN {X 0,Y 397.211,Z 295.632,A -85,B 0,C 180,E1 -11329.809,E2 -11329.809} C_VEL
LIN {X 0,Y 397.287,Z 295.622,A -85,B 0,C 180,E1 -11332.887,E2 -11332.887} C_VEL
LIN {X 0,Y 397.24,Z 295.626,A -85,B 0,C 180,E1 -11334.925,E2 -11334.925} C_VEL
LIN {X 0,Y 397.444,Z 295.599,A -85,B 0,C 180,E1 -11337.973,E2 -11337.973} C_VEL
LIN {X 0,Y 397.568,Z 295.59,A -85,B 0,C 180,E1 -11340,E2 -11340} C_VEL
LIN {X 0,Y 397.375,Z 295.614,A -85,B 0,C 180,E1 -11343.042,E2 -11343.042} C_VEL
LIN {X 0,Y 397.299,Z 295.62,A -85,B 0,C 180,E1 -11346.435,E2 -11346.435} C_VEL
LIN {X 0,Y 397.228,Z 295.63,A -85,B 0,C 180,E1 -11349.163,E2 -11349.163} C_VEL
LIN {X 0,Y 397.211,Z 295.632,A -85,B 0,C 180,E1 -11352.258,E2 -11352.258} C_VEL
LIN {X 0,Y 397.171,Z 295.637,A -85,B 0,C 180,E1 -11355.392,E2 -11355.392} C_VEL
LIN {X 0,Y 397.155,Z 295.641,A -85,B 0,C 180,E1 -11358.574,E2 -11358.574} C_VEL
LIN {X 0,Y 397.101,Z 295.646,A -85,B 0,C 180,E1 -11361.818,E2 -11361.818} C_VEL
LIN {X 0,Y 397.146,Z 295.639,A -85,B 0,C 180,E1 -11365.513,E2 -11365.513} C_VEL
LIN {X 0,Y 397.115,Z 295.641,A -85,B 0,C 180,E1 -11368.544,E2 -11368.544} C_VEL
LIN {X 0,Y 397.072,Z 295.648,A -85,B 0,C 180,E1 -11372.072,E2 -11372.072} C_VEL
LIN {X 0,Y 397.113,Z 295.643,A -85,B 0,C 180,E1 -11375.504,E2 -11375.504} C_VEL
LIN {X 0,Y 397.127,Z 295.643,A -85,B 0,C 180,E1 -11378.863,E2 -11378.863} C_VEL
LIN {X 0,Y 397.064,Z 295.652,A -85,B 0,C 180,E1 -11382.268,E2 -11382.268} C_VEL
LIN {X 0,Y 397.135,Z 295.941,A -85,B 0,C 180,E1 -11384.94,E2 -11384.94} C_VEL
LIN {X 0,Y 397.475,Z 299.149,A -85,B 0,C 180,E1 -11387.956,E2 -11387.956} C_VEL
LIN {X 0,Y 397.418,Z 301.96,A -85,B 0,C 180,E1 -11390.46,E2 -11390.46} C_VEL
LIN {X 0,Y 397.185,Z 306.47,A -85,B 0,C 180,E1 -11394.274,E2 -11394.274} C_VEL
LIN {X 0,Y 396.965,Z 309.486,A -85,B 0,C 180,E1 -11396.714,E2 -11396.714} C_VEL
LIN {X 0,Y 396.706,Z 314.028,A -85,B 0,C 180,E1 -11400.262,E2 -11400.262} C_VEL
LIN {X 0,Y 396.446,Z 318.967,A -85,B 0,C 180,E1 -11403.992,E2 -11403.992} C_VEL
LIN {X 0,Y 396.443,Z 319.137,A -85,B 0,C 180,E1 -11404.118,E2 -11404.118} C_VEL
LIN {X 0,Y 398.066,Z 324.374,A -85,B 0,C 180,E1 -11404.364,E2 -11404.364} C_VEL
LIN {X 0,Y 402.507,Z 338.135,A -85,B 0,C 180,E1 -11405.083,E2 -11405.083} C_VEL
LIN {X 0,Y 406.206,Z 352.451,A -85,B 0,C 180,E1 -11405.946,E2 -11405.946} C_VEL
LIN {X 0,Y 407.343,Z 357.576,A -85,B 0,C 180,E1 -11406.285,E2 -11406.285} C_VEL
LIN {X 0,Y 406.25,Z 371.742,A -85,B 0,C 180,E1 -11407.114,E2 -11407.114} C_VEL
LIN {X 0,Y 404.732,Z 386.597,A -85,B 0,C 180,E1 -11408.213,E2 -11408.213} C_VEL
LIN {X 0,Y 403.275,Z 400.092,A -85,B 0,C 180,E1 -11409.469,E2 -11409.469} C_VEL
LIN {X 0,Y 401.959,Z 411.543,A -85,B 0,C 180,E1 -11410.762,E2 -11410.762} C_VEL
LIN {X 0,Y 400.494,Z 423.494,A -85,B 0,C 180,E1 -11412.38,E2 -11412.38} C_VEL
LIN {X 0,Y 399.193,Z 434.333,A -85,B 0,C 180,E1 -11414.165,E2 -11414.165} C_VEL
LIN {X 0,Y 398.01,Z 444.014,A -85,B 0,C 180,E1 -11416.107,E2 -11416.107} C_VEL
LIN {X 0,Y 397.374,Z 450.788,A -85,B 0,C 180,E1 -11417.747,E2 -11417.747} C_VEL
LIN {X 0,Y 396.599,Z 457.762,A -85,B 0,C 180,E1 -11419.793,E2 -11419.793} C_VEL
LIN {X 0,Y 396.163,Z 463.243,A -85,B 0,C 180,E1 -11421.841,E2 -11421.841} C_VEL
LIN {X 0,Y 395.909,Z 467.382,A -85,B 0,C 180,E1 -11423.886,E2 -11423.886} C_VEL
LIN {X 0,Y 395.764,Z 470.292,A -85,B 0,C 180,E1 -11425.927,E2 -11425.927} C_VEL
LIN {X 0,Y 395.759,Z 472.043,A -85,B 0,C 180,E1 -11427.965,E2 -11427.965} C_VEL
LIN {X 0,Y 395.758,Z 472.655,A -85,B 0,C 180,E1 -11430,E2 -11430} C_VEL
LIN {X 0,Y 395.759,Z 472.09,A -85,B 0,C 180,E1 -11432.036,E2 -11432.036} C_VEL
LIN {X 0,Y 395.763,Z 470.401,A -85,B 0,C 180,E1 -11434.074,E2 -11434.074} C_VEL
LIN {X 0,Y 395.915,Z 467.329,A -85,B 0,C 180,E1 -11436.241,E2 -11436.241} C_VEL
LIN {X 0,Y 396.16,Z 463.468,A -85,B 0,C 180,E1 -11438.159,E2 -11438.159} C_VEL
LIN {X 0,Y 396.577,Z 458.058,A -85,B 0,C 180,E1 -11440.208,E2 -11440.208} C_VEL
LIN {X 0,Y 397.353,Z 451.163,A -85,B 0,C 180,E1 -11442.254,E2 -11442.254} C_VEL
LIN {X 0,Y 397.947,Z 444.472,A -85,B 0,C 180,E1 -11443.886,E2 -11443.886} C_VEL
LIN {X 0,Y 398.598,Z 438.929,A -85,B 0,C 180,E1 -11445.062,E2 -11445.062} C_VEL
LIN {X 0,Y 398.425,Z 435.538,A -85,B 0,C 180,E1 -11445.755,E2 -11445.755} C_VEL
LIN {X 0,Y 396.398,Z 429.807,A -85,B 0,C 180,E1 -11446.883,E2 -11446.883} C_VEL
LIN {X 0,Y 394.399,Z 423.718,A -85,B 0,C 180,E1 -11447.974,E2 -11447.974} C_VEL
LIN {X 0,Y 394.268,Z 419.629,A -85,B 0,C 180,E1 -11448.601,E2 -11448.601} C_VEL
LIN {X 0,Y 395.582,Z 408.924,A -85,B 0,C 180,E1 -11449.999,E2 -11449.999} C_VEL
LIN {X 0,Y 397.031,Z 397.248,A -85,B 0,C 180,E1 -11451.277,E2 -11451.277} C_VEL
LIN {X 0,Y 398.351,Z 384.663,A -85,B 0,C 180,E1 -11452.428,E2 -11452.428} C_VEL
LIN {X 0,Y 399.796,Z 371.279,A -85,B 0,C 180,E1 -11453.413,E2 -11453.413} C_VEL
LIN {X 0,Y 400.663,Z 358.28,A -85,B 0,C 180,E1 -11454.199,E2 -11454.199} C_VEL
LIN {X 0,Y 396.855,Z 342.742,A -85,B 0,C 180,E1 -11455.221,E2 -11455.221} C_VEL
LIN {X 0,Y 392.513,Z 328.512,A -85,B 0,C 180,E1 -11456.023,E2 -11456.023} C_VEL
LIN {X 0,Y 389.449,Z 319.725,A -85,B 0,C 180,E1 -11456.46,E2 -11456.46} C_VEL
LIN {X 0,Y 389.395,Z 319.214,A -85,B 0,C 180,E1 -11456.504,E2 -11456.504} C_VEL
LIN {X 0,Y 389.684,Z 314.654,A -85,B 0,C 180,E1 -11460.039,E2 -11460.039} C_VEL
LIN {X 0,Y 389.872,Z 311.251,A -85,B 0,C 180,E1 -11462.737,E2 -11462.737} C_VEL
LIN {X 0,Y 390.149,Z 307.47,A -85,B 0,C 180,E1 -11465.844,E2 -11465.844} C_VEL
LIN {X 0,Y 390.374,Z 303.46,A -85,B 0,C 180,E1 -11469.273,E2 -11469.273} C_VEL
LIN {X 0,Y 390.465,Z 300.659,A -85,B 0,C 180,E1 -11471.756,E2 -11471.756} C_VEL
LIN {X 0,Y 390.22,Z 297.627,A -85,B 0,C 180,E1 -11474.62,E2 -11474.62} C_VEL
LIN {X 0,Y 390.12,Z 296.868,A -85,B 0,C 180,E1 -11475.365,E2 -11475.365} C_VEL
LIN {X 0,Y 390.057,Z 296.526,A -85,B 0,C 180,E1 -11476.789,E2 -11476.789} C_VEL
LIN {X 0,Y 390.056,Z 296.522,A -85,B 0,C 180,E1 -11479.56,E2 -11479.56} C_VEL
LIN {X 0,Y 390.042,Z 296.527,A -85,B 0,C 180,E1 -11482.449,E2 -11482.449} C_VEL
LIN {X 0,Y 390.067,Z 296.525,A -85,B 0,C 180,E1 -11486.045,E2 -11486.045} C_VEL
LIN {X 0,Y 390.042,Z 296.526,A -85,B 0,C 180,E1 -11489.869,E2 -11489.869} C_VEL
LIN {X 0,Y 390.053,Z 296.521,A -85,B 0,C 180,E1 -11493.227,E2 -11493.227} C_VEL
LIN {X 0,Y 390.065,Z 296.523,A -85,B 0,C 180,E1 -11496.764,E2 -11496.764} C_VEL
LIN {X 0,Y 390.102,Z 296.519,A -85,B 0,C 180,E1 -11499.983,E2 -11499.983} C_VEL
LIN {X 0,Y 390.136,Z 296.512,A -85,B 0,C 180,E1 -11503.248,E2 -11503.248} C_VEL
LIN {X 0,Y 390.192,Z 296.503,A -85,B 0,C 180,E1 -11506.561,E2 -11506.561} C_VEL
LIN {X 0,Y 390.166,Z 296.51,A -85,B 0,C 180,E1 -11509.623,E2 -11509.623} C_VEL
LIN {X 0,Y 390.245,Z 296.5,A -85,B 0,C 180,E1 -11512.758,E2 -11512.758} C_VEL
LIN {X 0,Y 390.213,Z 296.503,A -85,B 0,C 180,E1 -11514.833,E2 -11514.833} C_VEL
LIN {X 0,Y 390.418,Z 296.477,A -85,B 0,C 180,E1 -11517.937,E2 -11517.937} C_VEL
LIN {X 0,Y 390.54,Z 296.465,A -85,B 0,C 180,E1 -11520,E2 -11520} C_VEL
LIN {X 0,Y 390.313,Z 296.493,A -85,B 0,C 180,E1 -11523.096,E2 -11523.096} C_VEL
LIN {X 0,Y 390.284,Z 296.497,A -85,B 0,C 180,E1 -11526.202,E2 -11526.202} C_VEL
LIN {X 0,Y 390.191,Z 296.509,A -85,B 0,C 180,E1 -11529.329,E2 -11529.329} C_VEL
LIN {X 0,Y 390.168,Z 296.511,A -85,B 0,C 180,E1 -11532.483,E2 -11532.483} C_VEL
LIN {X 0,Y 390.136,Z 296.514,A -85,B 0,C 180,E1 -11535.677,E2 -11535.677} C_VEL
LIN {X 0,Y 390.103,Z 296.517,A -85,B 0,C 180,E1 -11538.922,E2 -11538.922} C_VEL
LIN {X 0,Y 390.034,Z 296.525,A -85,B 0,C 180,E1 -11542.234,E2 -11542.234} C_VEL
LIN {X 0,Y 390.116,Z 296.516,A -85,B 0,C 180,E1 -11545.743,E2 -11545.743} C_VEL
LIN {X 0,Y 390.056,Z 296.528,A -85,B 0,C 180,E1 -11549.11,E2 -11549.11} C_VEL
LIN {X 0,Y 390.04,Z 296.531,A -85,B 0,C 180,E1 -11552.722,E2 -11552.722} C_VEL
LIN {X 0,Y 390.053,Z 296.53,A -85,B 0,C 180,E1 -11555.825,E2 -11555.825} C_VEL
LIN {X 0,Y 390.059,Z 296.528,A -85,B 0,C 180,E1 -11559.217,E2 -11559.217} C_VEL
LIN {X 0,Y 390.031,Z 296.529,A -85,B 0,C 180,E1 -11561.813,E2 -11561.813} C_VEL
LIN {X 0,Y 390.532,Z 299.431,A -85,B 0,C 180,E1 -11564.575,E2 -11564.575} C_VEL
LIN {X 0,Y 390.883,Z 302.922,A -85,B 0,C 180,E1 -11567.491,E2 -11567.491} C_VEL
LIN {X 0,Y 390.903,Z 305.694,A -85,B 0,C 180,E1 -11569.666,E2 -11569.666} C_VEL
LIN {X 0,Y 390.661,Z 309.233,A -85,B 0,C 180,E1 -11572.331,E2 -11572.331} C_VEL
LIN {X 0,Y 390.399,Z 312.683,A -85,B 0,C 180,E1 -11574.826,E2 -11574.826} C_VEL
LIN {X 0,Y 389.974,Z 317.948,A -85,B 0,C 180,E1 -11578.491,E2 -11578.491} C_VEL
LIN {X 0,Y 389.628,Z 323.337,A -85,B 0,C 180,E1 -11582.11,E2 -11582.11} C_VEL
LIN {X 0,Y 389.487,Z 325.53,A -85,B 0,C 180,E1 -11583.552,E2 -11583.552} C_VEL
LIN {X 0,Y 391.274,Z 331.478,A -85,B 0,C 180,E1 -11583.834,E2 -11583.834} C_VEL
LIN {X 0,Y 395.553,Z 345.354,A -85,B 0,C 180,E1 -11584.567,E2 -11584.567} C_VEL
LIN {X 0,Y 398.975,Z 359.388,A -85,B 0,C 180,E1 -11585.417,E2 -11585.417} C_VEL
LIN {X 0,Y 400.45,Z 367.624,A -85,B 0,C 180,E1 -11585.969,E2 -11585.969} C_VEL
LIN {X 0,Y 399.211,Z 381.709,A -85,B 0,C 180,E1 -11586.84,E2 -11586.84} C_VEL
LIN {X 0,Y 397.867,Z 394.396,A -85,B 0,C 180,E1 -11587.817,E2 -11587.817} C_VEL
LIN {X 0,Y 396.298,Z 407.809,A -85,B 0,C 180,E1 -11589.09,E2 -11589.09} C_VEL
LIN {X 0,Y 394.868,Z 419.502,A -85,B 0,C 180,E1 -11590.434,E2 -11590.434} C_VEL
LIN {X 0,Y 393.423,Z 431.174,A -85,B 0,C 180,E1 -11592.052,E2 -11592.052} C_VEL
LIN {X 0,Y 392.187,Z 440.554,A -85,B 0,C 180,E1 -11593.606,E2 -11593.606} C_VEL
LIN {X 0,Y 391.016,Z 449.783,A -85,B 0,C 180,E1 -11595.426,E2 -11595.426} C_VEL
LIN {X 0,Y 390.178,Z 457.458,A -85,B 0,C 180,E1 -11597.253,E2 -11597.253} C_VEL
LIN {X 0,Y 389.549,Z 463.821,A -85,B 0,C 180,E1 -11599.08,E2 -11599.08} C_VEL
LIN {X 0,Y 389.098,Z 469.67,A -85,B 0,C 180,E1 -11601.168,E2 -11601.168} C_VEL
LIN {X 0,Y 388.849,Z 473.146,A -85,B 0,C 180,E1 -11602.731,E2 -11602.731} C_VEL
LIN {X 0,Y 388.685,Z 476.658,A -85,B 0,C 180,E1 -11604.813,E2 -11604.813} C_VEL
LIN {X 0,Y 388.589,Z 478.968,A -85,B 0,C 180,E1 -11606.889,E2 -11606.889} C_VEL
LIN {X 0,Y 388.652,Z 480.13,A -85,B 0,C 180,E1 -11608.963,E2 -11608.963} C_VEL
LIN {X 0,Y 388.652,Z 480.129,A -85,B 0,C 180,E1 -11611.036,E2 -11611.036} C_VEL
LIN {X 0,Y 388.589,Z 478.96,A -85,B 0,C 180,E1 -11613.11,E2 -11613.11} C_VEL
LIN {X 0,Y 388.693,Z 476.646,A -85,B 0,C 180,E1 -11615.186,E2 -11615.186} C_VEL
LIN {X 0,Y 388.913,Z 473.137,A -85,B 0,C 180,E1 -11617.267,E2 -11617.267} C_VEL
LIN {X 0,Y 389.183,Z 468.34,A -85,B 0,C 180,E1 -11619.353,E2 -11619.353} C_VEL
LIN {X 0,Y 389.774,Z 462.129,A -85,B 0,C 180,E1 -11621.439,E2 -11621.439} C_VEL
LIN {X 0,Y 390.481,Z 454.325,A -85,B 0,C 180,E1 -11623.531,E2 -11623.531} C_VEL
LIN {X 0,Y 391.507,Z 446.026,A -85,B 0,C 180,E1 -11625.353,E2 -11625.353} C_VEL
LIN {X 0,Y 392.716,Z 436.025,A -85,B 0,C 180,E1 -11627.174,E2 -11627.174} C_VEL
LIN {X 0,Y 394.235,Z 424.665,A -85,B 0,C 180,E1 -11628.878,E2 -11628.878} C_VEL
LIN {X 0,Y 395.719,Z 412.456,A -85,B 0,C 180,E1 -11630.397,E2 -11630.397} C_VEL
LIN {X 0,Y 397.171,Z 400.029,A -85,B 0,C 180,E1 -11631.677,E2 -11631.677} C_VEL
LIN {X 0,Y 398.694,Z 386.415,A -85,B 0,C 180,E1 -11632.817,E2 -11632.817} C_VEL
LIN {X 0,Y 400.038,Z 372.908,A -85,B 0,C 180,E1 -11633.724,E2 -11633.724} C_VEL
LIN {X 0,Y 400.341,Z 366.534,A -85,B 0,C 180,E1 -11634.096,E2 -11634.096} C_VEL
LIN {X 0,Y 397.416,Z 352.797,A -85,B 0,C 180,E1 -11634.992,E2 -11634.992} C_VEL
LIN {X 0,Y 393.343,Z 337.826,A -85,B 0,C 180,E1 -11635.833,E2 -11635.833} C_VEL
LIN {X 0,Y 389.602,Z 326.432,A -85,B 0,C 180,E1 -11636.394,E2 -11636.394} C_VEL
LIN {X 0,Y 389.495,Z 325.506,A -85,B 0,C 180,E1 -11636.467,E2 -11636.467} C_VEL
LIN {X 0,Y 389.821,Z 320.089,A -85,B 0,C 180,E1 -11640.074,E2 -11640.074} C_VEL
LIN {X 0,Y 390.09,Z 316.246,A -85,B 0,C 180,E1 -11642.716,E2 -11642.716} C_VEL
LIN {X 0,Y 390.473,Z 311.715,A -85,B 0,C 180,E1 -11645.91,E2 -11645.91} C_VEL
LIN {X 0,Y 390.82,Z 307.005,A -85,B 0,C 180,E1 -11649.353,E2 -11649.353} C_VEL
LIN {X 0,Y 390.913,Z 303.952,A -85,B 0,C 180,E1 -11651.696,E2 -11651.696} C_VEL
LIN {X 0,Y 390.666,Z 300.441,A -85,B 0,C 180,E1 -11654.554,E2 -11654.554} C_VEL
LIN {X 0,Y 390.096,Z 296.942,A -85,B 0,C 180,E1 -11657.616,E2 -11657.616} C_VEL
LIN {X 0,Y 390.031,Z 296.53,A -85,B 0,C 180,E1 -11658.187,E2 -11658.187} C_VEL
LIN {X 0,Y 390.084,Z 296.521,A -85,B 0,C 180,E1 -11660.907,E2 -11660.907} C_VEL
LIN {X 0,Y 390.078,Z 296.526,A -85,B 0,C 180,E1 -11664.793,E2 -11664.793} C_VEL
LIN {X 0,Y 390.017,Z 296.533,A -85,B 0,C 180,E1 -11668.495,E2 -11668.495} C_VEL
LIN {X 0,Y 390.11,Z 296.52,A -85,B 0,C 180,E1 -11672.07,E2 -11672.07} C_VEL
LIN {X 0,Y 390.073,Z 296.525,A -85,B 0,C 180,E1 -11675.519,E2 -11675.519} C_VEL
LIN {X 0,Y 390.048,Z 296.526,A -85,B 0,C 180,E1 -11678.877,E2 -11678.877} C_VEL
LIN {X 0,Y 390.12,Z 296.514,A -85,B 0,C 180,E1 -11682.166,E2 -11682.166} C_VEL
LIN {X 0,Y 390.135,Z 296.511,A -85,B 0,C 180,E1 -11685.392,E2 -11685.392} C_VEL
LIN {X 0,Y 390.141,Z 296.511,A -85,B 0,C 180,E1 -11688.571,E2 -11688.571} C_VEL
LIN {X 0,Y 390.248,Z 296.499,A -85,B 0,C 180,E1 -11692.086,E2 -11692.086} C_VEL
LIN {X 0,Y 390.21,Z 296.501,A -85,B 0,C 180,E1 -11694.833,E2 -11694.833} C_VEL
LIN {X 0,Y 390.413,Z 296.474,A -85,B 0,C 180,E1 -11697.937,E2 -11697.937} C_VEL
LIN {X 0,Y 390.537,Z 296.465,A -85,B 0,C 180,E1 -11700,E2 -11700} C_VEL
LIN {X 0,Y 390.309,Z 296.494,A -85,B 0,C 180,E1 -11703.097,E2 -11703.097} C_VEL
LIN {X 0,Y 390.261,Z 296.499,A -85,B 0,C 180,E1 -11706.424,E2 -11706.424} C_VEL
LIN {X 0,Y 390.186,Z 296.509,A -85,B 0,C 180,E1 -11709.329,E2 -11709.329} C_VEL
LIN {X 0,Y 390.163,Z 296.511,A -85,B 0,C 180,E1 -11712.483,E2 -11712.483} C_VEL
LIN {X 0,Y 390.131,Z 296.514,A -85,B 0,C 180,E1 -11715.677,E2 -11715.677} C_VEL
LIN {X 0,Y 390.098,Z 296.518,A -85,B 0,C 180,E1 -11718.923,E2 -11718.923} C_VEL
LIN {X 0,Y 390.04,Z 296.524,A -85,B 0,C 180,E1 -11722.234,E2 -11722.234} C_VEL
LIN {X 0,Y 390.112,Z 296.517,A -85,B 0,C 180,E1 -11725.744,E2 -11725.744} C_VEL
LIN {X 0,Y 390.052,Z 296.523,A -85,B 0,C 180,E1 -11729.11,E2 -11729.11} C_VEL
LIN {X 0,Y 390.037,Z 296.522,A -85,B 0,C 180,E1 -11732.722,E2 -11732.722} C_VEL
LIN {X 0,Y 390.05,Z 296.522,A -85,B 0,C 180,E1 -11735.826,E2 -11735.826} C_VEL
LIN {X 0,Y 390.066,Z 296.523,A -85,B 0,C 180,E1 -11739.219,E2 -11739.219} C_VEL
LIN {X 0,Y 390.038,Z 296.527,A -85,B 0,C 180,E1 -11742.375,E2 -11742.375} C_VEL
LIN {X 0,Y 390.077,Z 296.755,A -85,B 0,C 180,E1 -11744.641,E2 -11744.641} C_VEL
LIN {X 0,Y 390.412,Z 299.799,A -85,B 0,C 180,E1 -11747.567,E2 -11747.567} C_VEL
LIN {X 0,Y 390.439,Z 302.025,A -85,B 0,C 180,E1 -11749.61,E2 -11749.61} C_VEL
LIN {X 0,Y 390.243,Z 305.219,A -85,B 0,C 180,E1 -11752.411,E2 -11752.411} C_VEL
LIN {X 0,Y 390.112,Z 308.034,A -85,B 0,C 180,E1 -11754.797,E2 -11754.797} C_VEL
LIN {X 0,Y 389.773,Z 312.582,A -85,B 0,C 180,E1 -11758.474,E2 -11758.474} C_VEL
LIN {X 0,Y 389.609,Z 315.616,A -85,B 0,C 180,E1 -11760.855,E2 -11760.855} C_VEL
LIN {X 0,Y 389.446,Z 319.385,A -85,B 0,C 180,E1 -11763.634,E2 -11763.634} C_VEL
LIN {X 0,Y 391.469,Z 325.467,A -85,B 0,C 180,E1 -11763.924,E2 -11763.924} C_VEL
LIN {X 0,Y 395.972,Z 339.684,A -85,B 0,C 180,E1 -11764.699,E2 -11764.699} C_VEL
LIN {X 0,Y 399.655,Z 353.977,A -85,B 0,C 180,E1 -11765.603,E2 -11765.603} C_VEL
LIN {X 0,Y 400.714,Z 359.123,A -85,B 0,C 180,E1 -11765.954,E2 -11765.954} C_VEL
LIN {X 0,Y 399.496,Z 373.896,A -85,B 0,C 180,E1 -11766.86,E2 -11766.86} C_VEL
LIN {X 0,Y 398.141,Z 386.672,A -85,B 0,C 180,E1 -11767.834,E2 -11767.834} C_VEL
LIN {X 0,Y 396.617,Z 400.166,A -85,B 0,C 180,E1 -11769.108,E2 -11769.108} C_VEL
LIN {X 0,Y 395.139,Z 412.294,A -85,B 0,C 180,E1 -11770.504,E2 -11770.504} C_VEL
LIN {X 0,Y 393.69,Z 423.567,A -85,B 0,C 180,E1 -11772.066,E2 -11772.066} C_VEL
LIN {X 0,Y 392.319,Z 434.405,A -85,B 0,C 180,E1 -11773.88,E2 -11773.88} C_VEL
LIN {X 0,Y 391.179,Z 443.307,A -85,B 0,C 180,E1 -11775.677,E2 -11775.677} C_VEL
LIN {X 0,Y 390.396,Z 450.859,A -85,B 0,C 180,E1 -11777.525,E2 -11777.525} C_VEL
LIN {X 0,Y 389.553,Z 457.833,A -85,B 0,C 180,E1 -11779.607,E2 -11779.607} C_VEL
LIN {X 0,Y 389.105,Z 463.314,A -85,B 0,C 180,E1 -11781.692,E2 -11781.692} C_VEL
LIN {X 0,Y 388.834,Z 467.452,A -85,B 0,C 180,E1 -11783.775,E2 -11783.775} C_VEL
LIN {X 0,Y 388.69,Z 470.362,A -85,B 0,C 180,E1 -11785.853,E2 -11785.853} C_VEL
LIN {X 0,Y 388.656,Z 472.112,A -85,B 0,C 180,E1 -11787.928,E2 -11787.928} C_VEL
LIN {X 0,Y 388.671,Z 472.724,A -85,B 0,C 180,E1 -11790,E2 -11790} C_VEL
LIN {X 0,Y 388.656,Z 472.159,A -85,B 0,C 180,E1 -11792.073,E2 -11792.073} C_VEL
LIN {X 0,Y 388.689,Z 470.47,A -85,B 0,C 180,E1 -11794.148,E2 -11794.148} C_VEL
LIN {X 0,Y 388.834,Z 467.618,A -85,B 0,C 180,E1 -11796.226,E2 -11796.226} C_VEL
LIN {X 0,Y 389.101,Z 463.536,A -85,B 0,C 180,E1 -11798.308,E2 -11798.308} C_VEL
LIN {X 0,Y 389.532,Z 458.126,A -85,B 0,C 180,E1 -11800.395,E2 -11800.395} C_VEL
LIN {X 0,Y 390.375,Z 451.231,A -85,B 0,C 180,E1 -11802.477,E2 -11802.477} C_VEL
LIN {X 0,Y 391.086,Z 443.856,A -85,B 0,C 180,E1 -11804.298,E2 -11804.298} C_VEL
LIN {X 0,Y 392.213,Z 434.893,A -85,B 0,C 180,E1 -11806.126,E2 -11806.126} C_VEL
LIN {X 0,Y 393.346,Z 425.792,A -85,B 0,C 180,E1 -11807.683,E2 -11807.683} C_VEL
LIN {X 0,Y 394.268,Z 419.629,A -85,B 0,C 180,E1 -11808.601,E2 -11808.601} C_VEL
LIN {X 0,Y 394.172,Z 415.488,A -85,B 0,C 180,E1 -11809.213,E2 -11809.213} C_VEL
LIN {X 0,Y 392.346,Z 408.659,A -85,B 0,C 180,E1 -11810.225,E2 -11810.225} C_VEL
LIN {X 0,Y 390.537,Z 401.496,A -85,B 0,C 180,E1 -11811.186,E2 -11811.186} C_VEL
LIN {X 0,Y 390.455,Z 396.781,A -85,B 0,C 180,E1 -11811.711,E2 -11811.711} C_VEL
LIN {X 0,Y 391.799,Z 384.726,A -85,B 0,C 180,E1 -11812.824,E2 -11812.824} C_VEL
LIN {X 0,Y 393.231,Z 371.896,A -85,B 0,C 180,E1 -11813.789,E2 -11813.789} C_VEL
LIN {X 0,Y 394.056,Z 359.622,A -85,B 0,C 180,E1 -11814.552,E2 -11814.552} C_VEL
LIN {X 0,Y 390.458,Z 344.677,A -85,B 0,C 180,E1 -11815.579,E2 -11815.579} C_VEL
LIN {X 0,Y 386.396,Z 331.182,A -85,B 0,C 180,E1 -11816.383,E2 -11816.383} C_VEL
LIN {X 0,Y 382.407,Z 319.63,A -85,B 0,C 180,E1 -11816.989,E2 -11816.989} C_VEL
LIN {X 0,Y 382.377,Z 319.242,A -85,B 0,C 180,E1 -11817.063,E2 -11817.063} C_VEL
LIN {X 0,Y 382.688,Z 314.336,A -85,B 0,C 180,E1 -11820.945,E2 -11820.945} C_VEL
LIN {X 0,Y 383.016,Z 309.808,A -85,B 0,C 180,E1 -11824.668,E2 -11824.668} C_VEL
LIN {X 0,Y 383.227,Z 305.985,A -85,B 0,C 180,E1 -11827.947,E2 -11827.947} C_VEL
LIN {X 0,Y 383.405,Z 303.745,A -85,B 0,C 180,E1 -11829.909,E2 -11829.909} C_VEL
LIN {X 0,Y 383.377,Z 300.702,A -85,B 0,C 180,E1 -11832.709,E2 -11832.709} C_VEL
LIN {X 0,Y 383.028,Z 297.572,A -85,B 0,C 180,E1 -11835.794,E2 -11835.794} C_VEL
LIN {X 0,Y 382.988,Z 297.407,A -85,B 0,C 180,E1 -11838.796,E2 -11838.796} C_VEL
LIN {X 0,Y 382.999,Z 297.406,A -85,B 0,C 180,E1 -11842.096,E2 -11842.096} C_VEL
LIN {X 0,Y 383.017,Z 297.403,A -85,B 0,C 180,E1 -11845.332,E2 -11845.332} C_VEL
LIN {X 0,Y 382.98,Z 297.406,A -85,B 0,C 180,E1 -11849.081,E2 -11849.081} C_VEL
LIN {X 0,Y 382.991,Z 297.403,A -85,B 0,C 180,E1 -11852.693,E2 -11852.693} C_VEL
LIN {X 0,Y 383.015,Z 297.4,A -85,B 0,C 180,E1 -11856.191,E2 -11856.191} C_VEL
LIN {X 0,Y 383.053,Z 297.395,A -85,B 0,C 180,E1 -11859.598,E2 -11859.598} C_VEL
LIN {X 0,Y 383.103,Z 297.39,A -85,B 0,C 180,E1 -11862.931,E2 -11862.931} C_VEL
LIN {X 0,Y 383.123,Z 297.384,A -85,B 0,C 180,E1 -11866.464,E2 -11866.464} C_VEL
LIN {X 0,Y 383.129,Z 297.387,A -85,B 0,C 180,E1 -11869.43,E2 -11869.43} C_VEL
LIN {X 0,Y 383.198,Z 297.379,A -85,B 0,C 180,E1 -11872.624,E2 -11872.624} C_VEL
LIN {X 0,Y 383.183,Z 297.379,A -85,B 0,C 180,E1 -11874.738,E2 -11874.738} C_VEL
LIN {X 0,Y 383.385,Z 297.353,A -85,B 0,C 180,E1 -11877.899,E2 -11877.899} C_VEL
LIN {X 0,Y 383.51,Z 297.34,A -85,B 0,C 180,E1 -11880,E2 -11880} C_VEL
LIN {X 0,Y 383.249,Z 297.373,A -85,B 0,C 180,E1 -11883.154,E2 -11883.154} C_VEL
LIN {X 0,Y 383.24,Z 297.373,A -85,B 0,C 180,E1 -11886.317,E2 -11886.317} C_VEL
LIN {X 0,Y 383.141,Z 297.386,A -85,B 0,C 180,E1 -11889.502,E2 -11889.502} C_VEL
LIN {X 0,Y 383.123,Z 297.389,A -85,B 0,C 180,E1 -11893.536,E2 -11893.536} C_VEL
LIN {X 0,Y 383.092,Z 297.39,A -85,B 0,C 180,E1 -11897.454,E2 -11897.454} C_VEL
LIN {X 0,Y 383.026,Z 297.398,A -85,B 0,C 180,E1 -11900.647,E2 -11900.647} C_VEL
LIN {X 0,Y 383.023,Z 297.398,A -85,B 0,C 180,E1 -11903.808,E2 -11903.808} C_VEL
LIN {X 0,Y 383.077,Z 297.395,A -85,B 0,C 180,E1 -11906.123,E2 -11906.123} C_VEL
LIN {X 0,Y 382.989,Z 297.407,A -85,B 0,C 180,E1 -11909.7,E2 -11909.7} C_VEL
LIN {X 0,Y 383.001,Z 297.41,A -85,B 0,C 180,E1 -11913.401,E2 -11913.401} C_VEL
LIN {X 0,Y 383.029,Z 297.405,A -85,B 0,C 180,E1 -11916.164,E2 -11916.164} C_VEL
LIN {X 0,Y 383.004,Z 297.406,A -85,B 0,C 180,E1 -11919.959,E2 -11919.959} C_VEL
LIN {X 0,Y 382.982,Z 297.407,A -85,B 0,C 180,E1 -11921.348,E2 -11921.348} C_VEL
LIN {X 0,Y 383.461,Z 300.132,A -85,B 0,C 180,E1 -11924.143,E2 -11924.143} C_VEL
LIN {X 0,Y 383.835,Z 303.567,A -85,B 0,C 180,E1 -11927.088,E2 -11927.088} C_VEL
LIN {X 0,Y 383.898,Z 305.629,A -85,B 0,C 180,E1 -11928.773,E2 -11928.773} C_VEL
LIN {X 0,Y 383.656,Z 309.772,A -85,B 0,C 180,E1 -11931.97,E2 -11931.97} C_VEL
LIN {X 0,Y 383.284,Z 314.385,A -85,B 0,C 180,E1 -11935.36,E2 -11935.36} C_VEL
LIN {X 0,Y 382.86,Z 319.649,A -85,B 0,C 180,E1 -11939.07,E2 -11939.07} C_VEL
LIN {X 0,Y 382.484,Z 325.444,A -85,B 0,C 180,E1 -11943.017,E2 -11943.017} C_VEL
LIN {X 0,Y 384.145,Z 331.05,A -85,B 0,C 180,E1 -11943.302,E2 -11943.302} C_VEL
LIN {X 0,Y 388.69,Z 345.575,A -85,B 0,C 180,E1 -11944.096,E2 -11944.096} C_VEL
LIN {X 0,Y 392.245,Z 359.984,A -85,B 0,C 180,E1 -11945.002,E2 -11945.002} C_VEL
LIN {X 0,Y 393.834,Z 369.158,A -85,B 0,C 180,E1 -11945.638,E2 -11945.638} C_VEL
LIN {X 0,Y 392.488,Z 383.48,A -85,B 0,C 180,E1 -11946.565,E2 -11946.565} C_VEL
LIN {X 0,Y 390.903,Z 397.183,A -85,B 0,C 180,E1 -11947.678,E2 -11947.678} C_VEL
LIN {X 0,Y 389.332,Z 410.093,A -85,B 0,C 180,E1 -11948.975,E2 -11948.975} C_VEL
LIN {X 0,Y 387.869,Z 421.265,A -85,B 0,C 180,E1 -11950.324,E2 -11950.324} C_VEL
LIN {X 0,Y 386.364,Z 432.739,A -85,B 0,C 180,E1 -11951.987,E2 -11951.987} C_VEL
LIN {X 0,Y 385.123,Z 441.923,A -85,B 0,C 180,E1 -11953.569,E2 -11953.569} C_VEL
LIN {X 0,Y 383.963,Z 450.93,A -85,B 0,C 180,E1 -11955.423,E2 -11955.423} C_VEL
LIN {X 0,Y 383.099,Z 458.4,A -85,B 0,C 180,E1 -11957.282,E2 -11957.282} C_VEL
LIN {X 0,Y 382.533,Z 463.753,A -85,B 0,C 180,E1 -11958.877,E2 -11958.877} C_VEL
LIN {X 0,Y 382.026,Z 469.601,A -85,B 0,C 180,E1 -11961.003,E2 -11961.003} C_VEL
LIN {X 0,Y 381.797,Z 473.077,A -85,B 0,C 180,E1 -11962.596,E2 -11962.596} C_VEL
LIN {X 0,Y 381.594,Z 476.589,A -85,B 0,C 180,E1 -11964.716,E2 -11964.716} C_VEL
LIN {X 0,Y 381.502,Z 478.899,A -85,B 0,C 180,E1 -11966.832,E2 -11966.832} C_VEL
LIN {X 0,Y 381.55,Z 480.061,A -85,B 0,C 180,E1 -11968.944,E2 -11968.944} C_VEL
LIN {X 0,Y 381.55,Z 480.06,A -85,B 0,C 180,E1 -11971.055,E2 -11971.055} C_VEL
LIN {X 0,Y 381.502,Z 478.89,A -85,B 0,C 180,E1 -11973.168,E2 -11973.168} C_VEL
LIN {X 0,Y 381.605,Z 476.576,A -85,B 0,C 180,E1 -11975.283,E2 -11975.283} C_VEL
LIN {X 0,Y 381.834,Z 473.067,A -85,B 0,C 180,E1 -11977.402,E2 -11977.402} C_VEL
LIN {X 0,Y 382.113,Z 468.27,A -85,B 0,C 180,E1 -11979.528,E2 -11979.528} C_VEL
LIN {X 0,Y 382.752,Z 462.058,A -85,B 0,C 180,E1 -11981.652,E2 -11981.652} C_VEL
LIN {X 0,Y 383.524,Z 454.254,A -85,B 0,C 180,E1 -11983.781,E2 -11983.781} C_VEL
LIN {X 0,Y 384.599,Z 445.955,A -85,B 0,C 180,E1 -11985.636,E2 -11985.636} C_VEL
LIN {X 0,Y 385.889,Z 435.954,A -85,B 0,C 180,E1 -11987.487,E2 -11987.487} C_VEL
LIN {X 0,Y 387.336,Z 425.724,A -85,B 0,C 180,E1 -11989.062,E2 -11989.062} C_VEL
LIN {X 0,Y 388.894,Z 413.532,A -85,B 0,C 180,E1 -11990.633,E2 -11990.633} C_VEL
LIN {X 0,Y 390.551,Z 399.955,A -85,B 0,C 180,E1 -11992.064,E2 -11992.064} C_VEL
LIN {X 0,Y 392.139,Z 386.341,A -85,B 0,C 180,E1 -11993.221,E2 -11993.221} C_VEL
LIN {X 0,Y 393.533,Z 372.558,A -85,B 0,C 180,E1 -11994.16,E2 -11994.16} C_VEL
LIN {X 0,Y 393.723,Z 367.781,A -85,B 0,C 180,E1 -11994.446,E2 -11994.446} C_VEL
LIN {X 0,Y 390.635,Z 353.24,A -85,B 0,C 180,E1 -11995.432,E2 -11995.432} C_VEL
LIN {X 0,Y 386.767,Z 339.057,A -85,B 0,C 180,E1 -11996.264,E2 -11996.264} C_VEL
LIN {X 0,Y 382.57,Z 326.231,A -85,B 0,C 180,E1 -11996.92,E2 -11996.92} C_VEL
LIN {X 0,Y 382.481,Z 325.45,A -85,B 0,C 180,E1 -11996.982,E2 -11996.982} C_VEL
LIN {X 0,Y 382.859,Z 319.675,A -85,B 0,C 180,E1 -12000.929,E2 -12000.929} C_VEL
LIN {X 0,Y 383.285,Z 314.435,A -85,B 0,C 180,E1 -12004.639,E2 -12004.639} C_VEL
LIN {X 0,Y 383.653,Z 309.815,A -85,B 0,C 180,E1 -12008.029,E2 -12008.029} C_VEL
LIN {X 0,Y 383.898,Z 305.652,A -85,B 0,C 180,E1 -12011.226,E2 -12011.226} C_VEL
LIN {X 0,Y 383.741,Z 302.136,A -85,B 0,C 180,E1 -12014.101,E2 -12014.101} C_VEL
LIN {X 0,Y 383.164,Z 298.566,A -85,B 0,C 180,E1 -12017.262,E2 -12017.262} C_VEL
LIN {X 0,Y 382.985,Z 297.407,A -85,B 0,C 180,E1 -12018.795,E2 -12018.795} C_VEL
LIN {X 0,Y 382.993,Z 297.406,A -85,B 0,C 180,E1 -12022.096,E2 -12022.096} C_VEL
LIN {X 0,Y 383.011,Z 297.405,A -85,B 0,C 180,E1 -12025.332,E2 -12025.332} C_VEL
LIN {X 0,Y 382.976,Z 297.411,A -85,B 0,C 180,E1 -12029.081,E2 -12029.081} C_VEL
LIN {X 0,Y 383.049,Z 297.399,A -85,B 0,C 180,E1 -12032.698,E2 -12032.698} C_VEL
LIN {X 0,Y 383.026,Z 297.398,A -85,B 0,C 180,E1 -12036.192,E2 -12036.192} C_VEL
LIN {X 0,Y 383.048,Z 297.396,A -85,B 0,C 180,E1 -12039.598,E2 -12039.598} C_VEL
LIN {X 0,Y 383.097,Z 297.389,A -85,B 0,C 180,E1 -12042.931,E2 -12042.931} C_VEL
LIN {X 0,Y 383.117,Z 297.389,A -85,B 0,C 180,E1 -12046.464,E2 -12046.464} C_VEL
LIN {X 0,Y 383.124,Z 297.389,A -85,B 0,C 180,E1 -12049.43,E2 -12049.43} C_VEL
LIN {X 0,Y 383.193,Z 297.379,A -85,B 0,C 180,E1 -12052.624,E2 -12052.624} C_VEL
LIN {X 0,Y 383.18,Z 297.377,A -85,B 0,C 180,E1 -12054.738,E2 -12054.738} C_VEL
LIN {X 0,Y 383.38,Z 297.35,A -85,B 0,C 180,E1 -12057.899,E2 -12057.899} C_VEL
LIN {X 0,Y 383.507,Z 297.341,A -85,B 0,C 180,E1 -12060,E2 -12060} C_VEL
LIN {X 0,Y 383.245,Z 297.373,A -85,B 0,C 180,E1 -12063.154,E2 -12063.154} C_VEL
LIN {X 0,Y 383.227,Z 297.375,A -85,B 0,C 180,E1 -12066.41,E2 -12066.41} C_VEL
LIN {X 0,Y 383.136,Z 297.386,A -85,B 0,C 180,E1 -12069.503,E2 -12069.503} C_VEL
LIN {X 0,Y 383.118,Z 297.389,A -85,B 0,C 180,E1 -12073.536,E2 -12073.536} C_VEL
LIN {X 0,Y 383.087,Z 297.388,A -85,B 0,C 180,E1 -12077.455,E2 -12077.455} C_VEL
LIN {X 0,Y 383.024,Z 297.397,A -85,B 0,C 180,E1 -12080.648,E2 -12080.648} C_VEL
LIN {X 0,Y 383.027,Z 297.398,A -85,B 0,C 180,E1 -12083.808,E2 -12083.808} C_VEL
LIN {X 0,Y 383.05,Z 297.395,A -85,B 0,C 180,E1 -12087.303,E2 -12087.303} C_VEL
LIN {X 0,Y 382.977,Z 297.402,A -85,B 0,C 180,E1 -12090.919,E2 -12090.919} C_VEL
LIN {X 0,Y 383.012,Z 297.398,A -85,B 0,C 180,E1 -12094.669,E2 -12094.669} C_VEL
LIN {X 0,Y 382.995,Z 297.403,A -85,B 0,C 180,E1 -12097.905,E2 -12097.905} C_VEL
LIN {X 0,Y 382.979,Z 297.407,A -85,B 0,C 180,E1 -12101.348,E2 -12101.348} C_VEL
LIN {X 0,Y 383.009,Z 297.547,A -85,B 0,C 180,E1 -12104.307,E2 -12104.307} C_VEL
LIN {X 0,Y 383.362,Z 300.576,A -85,B 0,C 180,E1 -12107.29,E2 -12107.29} C_VEL
LIN {X 0,Y 383.387,Z 303.591,A -85,B 0,C 180,E1 -12110.09,E2 -12110.09} C_VEL
LIN {X 0,Y 383.116,Z 307.823,A -85,B 0,C 180,E1 -12113.819,E2 -12113.819} C_VEL
LIN {X 0,Y 382.864,Z 311.132,A -85,B 0,C 180,E1 -12116.587,E2 -12116.587} C_VEL
LIN {X 0,Y 382.59,Z 315.681,A -85,B 0,C 180,E1 -12120.267,E2 -12120.267} C_VEL
LIN {X 0,Y 382.387,Z 319.285,A -85,B 0,C 180,E1 -12123.092,E2 -12123.092} C_VEL
LIN {X 0,Y 384.237,Z 324.999,A -85,B 0,C 180,E1 -12123.381,E2 -12123.381} C_VEL
LIN {X 0,Y 388.865,Z 338.967,A -85,B 0,C 180,E1 -12124.172,E2 -12124.172} C_VEL
LIN {X 0,Y 392.521,Z 352.888,A -85,B 0,C 180,E1 -12125.066,E2 -12125.066} C_VEL
LIN {X 0,Y 394.003,Z 359.565,A -85,B 0,C 180,E1 -12125.541,E2 -12125.541} C_VEL
LIN {X 0,Y 393.232,Z 371.096,A -85,B 0,C 180,E1 -12126.255,E2 -12126.255} C_VEL
LIN {X 0,Y 391.71,Z 385.186,A -85,B 0,C 180,E1 -12127.311,E2 -12127.311} C_VEL
LIN {X 0,Y 390.115,Z 398.986,A -85,B 0,C 180,E1 -12128.605,E2 -12128.605} C_VEL
LIN {X 0,Y 388.674,Z 410.372,A -85,B 0,C 180,E1 -12129.907,E2 -12129.907} C_VEL
LIN {X 0,Y 387.15,Z 421.866,A -85,B 0,C 180,E1 -12131.478,E2 -12131.478} C_VEL
LIN {X 0,Y 385.805,Z 431.541,A -85,B 0,C 180,E1 -12133.055,E2 -12133.055} C_VEL
LIN {X 0,Y 384.528,Z 441.025,A -85,B 0,C 180,E1 -12134.904,E2 -12134.904} C_VEL
LIN {X 0,Y 383.537,Z 448.922,A -85,B 0,C 180,E1 -12136.759,E2 -12136.759} C_VEL
LIN {X 0,Y 382.933,Z 454.615,A -85,B 0,C 180,E1 -12138.353,E2 -12138.353} C_VEL
LIN {X 0,Y 382.291,Z 460.82,A -85,B 0,C 180,E1 -12140.477,E2 -12140.477} C_VEL
LIN {X 0,Y 381.858,Z 465.613,A -85,B 0,C 180,E1 -12142.598,E2 -12142.598} C_VEL
LIN {X 0,Y 381.672,Z 469.125,A -85,B 0,C 180,E1 -12144.718,E2 -12144.718} C_VEL
LIN {X 0,Y 381.54,Z 471.449,A -85,B 0,C 180,E1 -12146.833,E2 -12146.833} C_VEL
LIN {X 0,Y 381.557,Z 472.635,A -85,B 0,C 180,E1 -12148.945,E2 -12148.945} C_VEL
LIN {X 0,Y 381.557,Z 472.65,A -85,B 0,C 180,E1 -12151.056,E2 -12151.056} C_VEL
LIN {X 0,Y 381.54,Z 471.525,A -85,B 0,C 180,E1 -12153.168,E2 -12153.168} C_VEL
LIN {X 0,Y 381.669,Z 469.261,A -85,B 0,C 180,E1 -12155.283,E2 -12155.283} C_VEL
LIN {X 0,Y 381.858,Z 465.805,A -85,B 0,C 180,E1 -12157.402,E2 -12157.402} C_VEL
LIN {X 0,Y 382.269,Z 461.073,A -85,B 0,C 180,E1 -12159.524,E2 -12159.524} C_VEL
LIN {X 0,Y 382.915,Z 454.944,A -85,B 0,C 180,E1 -12161.648,E2 -12161.648} C_VEL
LIN {X 0,Y 383.623,Z 448.286,A -85,B 0,C 180,E1 -12163.508,E2 -12163.508} C_VEL
LIN {X 0,Y 384.635,Z 440.24,A -85,B 0,C 180,E1 -12165.364,E2 -12165.364} C_VEL
LIN {X 0,Y 385.957,Z 430.589,A -85,B 0,C 180,E1 -12167.212,E2 -12167.212} C_VEL
LIN {X 0,Y 387.411,Z 420.407,A -85,B 0,C 180,E1 -12168.833,E2 -12168.833} C_VEL
LIN {X 0,Y 388.872,Z 408.989,A -85,B 0,C 180,E1 -12170.359,E2 -12170.359} C_VEL
LIN {X 0,Y 390.455,Z 396.781,A -85,B 0,C 180,E1 -12171.711,E2 -12171.711} C_VEL
LIN {X 0,Y 390.406,Z 392.014,A -85,B 0,C 180,E1 -12172.217,E2 -12172.217} C_VEL
LIN {X 0,Y 388.732,Z 384.176,A -85,B 0,C 180,E1 -12173.079,E2 -12173.079} C_VEL
LIN {X 0,Y 386.998,Z 376.09,A -85,B 0,C 180,E1 -12173.88,E2 -12173.88} C_VEL
LIN {X 0,Y 386.838,Z 370.869,A -85,B 0,C 180,E1 -12174.285,E2 -12174.285} C_VEL
LIN {X 0,Y 387.576,Z 362.405,A -85,B 0,C 180,E1 -12174.817,E2 -12174.817} C_VEL
LIN {X 0,Y 385.324,Z 351.643,A -85,B 0,C 180,E1 -12175.608,E2 -12175.608} C_VEL
LIN {X 0,Y 381.253,Z 336.74,A -85,B 0,C 180,E1 -12176.579,E2 -12176.579} C_VEL
LIN {X 0,Y 375.943,Z 321.746,A -85,B 0,C 180,E1 -12177.442,E2 -12177.442} C_VEL
LIN {X 0,Y 375.358,Z 319.37,A -85,B 0,C 180,E1 -12177.563,E2 -12177.563} C_VEL
LIN {X 0,Y 375.617,Z 315.601,A -85,B 0,C 180,E1 -12180.606,E2 -12180.606} C_VEL
LIN {X 0,Y 375.974,Z 310.747,A -85,B 0,C 180,E1 -12184.666,E2 -12184.666} C_VEL
LIN {X 0,Y 376.236,Z 306.537,A -85,B 0,C 180,E1 -12188.321,E2 -12188.321} C_VEL
LIN {X 0,Y 376.395,Z 303.785,A -85,B 0,C 180,E1 -12190.807,E2 -12190.807} C_VEL
LIN {X 0,Y 376.285,Z 300.775,A -85,B 0,C 180,E1 -12193.714,E2 -12193.714} C_VEL
LIN {X 0,Y 375.94,Z 298.287,A -85,B 0,C 180,E1 -12196.235,E2 -12196.235} C_VEL
LIN {X 0,Y 375.988,Z 298.275,A -85,B 0,C 180,E1 -12200.029,E2 -12200.029} C_VEL
LIN {X 0,Y 375.963,Z 298.283,A -85,B 0,C 180,E1 -12203.495,E2 -12203.495} C_VEL
LIN {X 0,Y 375.959,Z 298.282,A -85,B 0,C 180,E1 -12205.888,E2 -12205.888} C_VEL
LIN {X 0,Y 375.96,Z 298.281,A -85,B 0,C 180,E1 -12209.687,E2 -12209.687} C_VEL
LIN {X 0,Y 375.932,Z 298.28,A -85,B 0,C 180,E1 -12213.341,E2 -12213.341} C_VEL
LIN {X 0,Y 375.975,Z 298.279,A -85,B 0,C 180,E1 -12216.887,E2 -12216.887} C_VEL
LIN {X 0,Y 375.996,Z 298.273,A -85,B 0,C 180,E1 -12220.339,E2 -12220.339} C_VEL
LIN {X 0,Y 376.026,Z 298.268,A -85,B 0,C 180,E1 -12223.719,E2 -12223.719} C_VEL
LIN {X 0,Y 376.101,Z 298.257,A -85,B 0,C 180,E1 -12227.042,E2 -12227.042} C_VEL
LIN {X 0,Y 376.111,Z 298.26,A -85,B 0,C 180,E1 -12230.318,E2 -12230.318} C_VEL
LIN {X 0,Y 376.199,Z 298.25,A -85,B 0,C 180,E1 -12233.564,E2 -12233.564} C_VEL
LIN {X 0,Y 376.351,Z 298.229,A -85,B 0,C 180,E1 -12237.859,E2 -12237.859} C_VEL
LIN {X 0,Y 376.479,Z 298.216,A -85,B 0,C 180,E1 -12240,E2 -12240} C_VEL
LIN {X 0,Y 376.187,Z 298.252,A -85,B 0,C 180,E1 -12243.213,E2 -12243.213} C_VEL
LIN {X 0,Y 376.199,Z 298.25,A -85,B 0,C 180,E1 -12246.436,E2 -12246.436} C_VEL
LIN {X 0,Y 376.111,Z 298.261,A -85,B 0,C 180,E1 -12249.682,E2 -12249.682} C_VEL
LIN {X 0,Y 376.087,Z 298.266,A -85,B 0,C 180,E1 -12253.658,E2 -12253.658} C_VEL
LIN {X 0,Y 376.041,Z 298.268,A -85,B 0,C 180,E1 -12257.607,E2 -12257.607} C_VEL
LIN {X 0,Y 375.976,Z 298.277,A -85,B 0,C 180,E1 -12260.832,E2 -12260.832} C_VEL
LIN {X 0,Y 375.987,Z 298.277,A -85,B 0,C 180,E1 -12264.282,E2 -12264.282} C_VEL
LIN {X 0,Y 376.017,Z 298.273,A -85,B 0,C 180,E1 -12266.652,E2 -12266.652} C_VEL
LIN {X 0,Y 375.962,Z 298.284,A -85,B 0,C 180,E1 -12270.313,E2 -12270.313} C_VEL
LIN {X 0,Y 375.958,Z 298.287,A -85,B 0,C 180,E1 -12274.112,E2 -12274.112} C_VEL
LIN {X 0,Y 375.951,Z 298.288,A -85,B 0,C 180,E1 -12276.741,E2 -12276.741} C_VEL
LIN {X 0,Y 375.984,Z 298.281,A -85,B 0,C 180,E1 -12279.97,E2 -12279.97} C_VEL
LIN {X 0,Y 375.969,Z 298.614,A -85,B 0,C 180,E1 -12281.607,E2 -12281.607} C_VEL
LIN {X 0,Y 376.626,Z 302.463,A -85,B 0,C 180,E1 -12285.161,E2 -12285.161} C_VEL
LIN {X 0,Y 376.867,Z 306.084,A -85,B 0,C 180,E1 -12288.24,E2 -12288.24} C_VEL
LIN {X 0,Y 376.749,Z 309.074,A -85,B 0,C 180,E1 -12290.636,E2 -12290.636} C_VEL
LIN {X 0,Y 376.463,Z 312.666,A -85,B 0,C 180,E1 -12293.393,E2 -12293.393} C_VEL
LIN {X 0,Y 376.155,Z 316.069,A -85,B 0,C 180,E1 -12295.909,E2 -12295.909} C_VEL
LIN {X 0,Y 375.751,Z 321.33,A -85,B 0,C 180,E1 -12299.668,E2 -12299.668} C_VEL
LIN {X 0,Y 375.486,Z 325.603,A -85,B 0,C 180,E1 -12302.505,E2 -12302.505} C_VEL
LIN {X 0,Y 377.33,Z 331.364,A -85,B 0,C 180,E1 -12302.789,E2 -12302.789} C_VEL
LIN {X 0,Y 382.097,Z 346.659,A -85,B 0,C 180,E1 -12303.661,E2 -12303.661} C_VEL
LIN {X 0,Y 385.559,Z 360.864,A -85,B 0,C 180,E1 -12304.591,E2 -12304.591} C_VEL
LIN {X 0,Y 387.281,Z 370.091,A -85,B 0,C 180,E1 -12305.261,E2 -12305.261} C_VEL
LIN {X 0,Y 385.954,Z 383.651,A -85,B 0,C 180,E1 -12306.163,E2 -12306.163} C_VEL
LIN {X 0,Y 384.33,Z 397.117,A -85,B 0,C 180,E1 -12307.275,E2 -12307.275} C_VEL
LIN {X 0,Y 382.665,Z 410.026,A -85,B 0,C 180,E1 -12308.591,E2 -12308.591} C_VEL
LIN {X 0,Y 381.031,Z 421.949,A -85,B 0,C 180,E1 -12310.063,E2 -12310.063} C_VEL
LIN {X 0,Y 379.564,Z 432.671,A -85,B 0,C 180,E1 -12311.653,E2 -12311.653} C_VEL
LIN {X 0,Y 378.261,Z 441.855,A -85,B 0,C 180,E1 -12313.262,E2 -12313.262} C_VEL
LIN {X 0,Y 377.025,Z 450.862,A -85,B 0,C 180,E1 -12315.149,E2 -12315.149} C_VEL
LIN {X 0,Y 376.106,Z 458.332,A -85,B 0,C 180,E1 -12317.042,E2 -12317.042} C_VEL
LIN {X 0,Y 375.524,Z 463.685,A -85,B 0,C 180,E1 -12318.667,E2 -12318.667} C_VEL
LIN {X 0,Y 374.955,Z 469.533,A -85,B 0,C 180,E1 -12320.832,E2 -12320.832} C_VEL
LIN {X 0,Y 374.712,Z 473.009,A -85,B 0,C 180,E1 -12322.456,E2 -12322.456} C_VEL
LIN {X 0,Y 374.509,Z 476.521,A -85,B 0,C 180,E1 -12324.616,E2 -12324.616} C_VEL
LIN {X 0,Y 374.419,Z 478.83,A -85,B 0,C 180,E1 -12326.772,E2 -12326.772} C_VEL
LIN {X 0,Y 374.449,Z 479.992,A -85,B 0,C 180,E1 -12328.924,E2 -12328.924} C_VEL
LIN {X 0,Y 374.449,Z 479.991,A -85,B 0,C 180,E1 -12331.075,E2 -12331.075} C_VEL
LIN {X 0,Y 374.419,Z 478.821,A -85,B 0,C 180,E1 -12333.228,E2 -12333.228} C_VEL
LIN {X 0,Y 374.521,Z 476.507,A -85,B 0,C 180,E1 -12335.383,E2 -12335.383} C_VEL
LIN {X 0,Y 374.741,Z 472.996,A -85,B 0,C 180,E1 -12337.543,E2 -12337.543} C_VEL
LIN {X 0,Y 375.065,Z 468.199,A -85,B 0,C 180,E1 -12339.708,E2 -12339.708} C_VEL
LIN {X 0,Y 375.742,Z 461.987,A -85,B 0,C 180,E1 -12341.873,E2 -12341.873} C_VEL
LIN {X 0,Y 376.577,Z 454.183,A -85,B 0,C 180,E1 -12344.04,E2 -12344.04} C_VEL
LIN {X 0,Y 377.703,Z 445.883,A -85,B 0,C 180,E1 -12345.929,E2 -12345.929} C_VEL
LIN {X 0,Y 379.079,Z 435.882,A -85,B 0,C 180,E1 -12347.812,E2 -12347.812} C_VEL
LIN {X 0,Y 380.67,Z 424.774,A -85,B 0,C 180,E1 -12349.541,E2 -12349.541} C_VEL
LIN {X 0,Y 382.345,Z 412.31,A -85,B 0,C 180,E1 -12351.144,E2 -12351.144} C_VEL
LIN {X 0,Y 383.943,Z 399.882,A -85,B 0,C 180,E1 -12352.464,E2 -12352.464} C_VEL
LIN {X 0,Y 385.62,Z 386.267,A -85,B 0,C 180,E1 -12353.637,E2 -12353.637} C_VEL
LIN {X 0,Y 387.062,Z 372.365,A -85,B 0,C 180,E1 -12354.598,E2 -12354.598} C_VEL
LIN {X 0,Y 387.128,Z 368.976,A -85,B 0,C 180,E1 -12354.809,E2 -12354.809} C_VEL
LIN {X 0,Y 384.015,Z 354.303,A -85,B 0,C 180,E1 -12355.848,E2 -12355.848} C_VEL
LIN {X 0,Y 380.184,Z 340.136,A -85,B 0,C 180,E1 -12356.717,E2 -12356.717} C_VEL
LIN {X 0,Y 375.512,Z 325.996,A -85,B 0,C 180,E1 -12357.471,E2 -12357.471} C_VEL
LIN {X 0,Y 375.443,Z 325.399,A -85,B 0,C 180,E1 -12357.514,E2 -12357.514} C_VEL
LIN {X 0,Y 375.79,Z 320.896,A -85,B 0,C 180,E1 -12360.651,E2 -12360.651} C_VEL
LIN {X 0,Y 376.156,Z 316.114,A -85,B 0,C 180,E1 -12364.09,E2 -12364.09} C_VEL
LIN {X 0,Y 376.465,Z 312.625,A -85,B 0,C 180,E1 -12366.682,E2 -12366.682} C_VEL
LIN {X 0,Y 376.765,Z 309.107,A -85,B 0,C 180,E1 -12369.361,E2 -12369.361} C_VEL
LIN {X 0,Y 376.858,Z 305.596,A -85,B 0,C 180,E1 -12372.171,E2 -12372.171} C_VEL
LIN {X 0,Y 376.586,Z 302.091,A -85,B 0,C 180,E1 -12375.166,E2 -12375.166} C_VEL
LIN {X 0,Y 375.965,Z 298.588,A -85,B 0,C 180,E1 -12378.392,E2 -12378.392} C_VEL
LIN {X 0,Y 375.956,Z 298.282,A -85,B 0,C 180,E1 -12380.537,E2 -12380.537} C_VEL
LIN {X 0,Y 375.957,Z 298.284,A -85,B 0,C 180,E1 -12383.495,E2 -12383.495} C_VEL
LIN {X 0,Y 375.953,Z 298.285,A -85,B 0,C 180,E1 -12385.888,E2 -12385.888} C_VEL
LIN {X 0,Y 375.958,Z 298.285,A -85,B 0,C 180,E1 -12389.687,E2 -12389.687} C_VEL
LIN {X 0,Y 376.013,Z 298.274,A -85,B 0,C 180,E1 -12393.347,E2 -12393.347} C_VEL
LIN {X 0,Y 375.989,Z 298.276,A -85,B 0,C 180,E1 -12396.888,E2 -12396.888} C_VEL
LIN {X 0,Y 375.99,Z 298.275,A -85,B 0,C 180,E1 -12400.339,E2 -12400.339} C_VEL
LIN {X 0,Y 376.021,Z 298.271,A -85,B 0,C 180,E1 -12403.719,E2 -12403.719} C_VEL
LIN {X 0,Y 376.096,Z 298.262,A -85,B 0,C 180,E1 -12407.042,E2 -12407.042} C_VEL
LIN {X 0,Y 376.106,Z 298.261,A -85,B 0,C 180,E1 -12410.318,E2 -12410.318} C_VEL
LIN {X 0,Y 376.194,Z 298.251,A -85,B 0,C 180,E1 -12413.564,E2 -12413.564} C_VEL
LIN {X 0,Y 376.346,Z 298.226,A -85,B 0,C 180,E1 -12417.86,E2 -12417.86} C_VEL
LIN {X 0,Y 376.476,Z 298.217,A -85,B 0,C 180,E1 -12420,E2 -12420} C_VEL
LIN {X 0,Y 376.183,Z 298.253,A -85,B 0,C 180,E1 -12423.213,E2 -12423.213} C_VEL
LIN {X 0,Y 376.194,Z 298.251,A -85,B 0,C 180,E1 -12426.436,E2 -12426.436} C_VEL
LIN {X 0,Y 376.106,Z 298.261,A -85,B 0,C 180,E1 -12429.682,E2 -12429.682} C_VEL
LIN {X 0,Y 376.082,Z 298.266,A -85,B 0,C 180,E1 -12433.658,E2 -12433.658} C_VEL
LIN {X 0,Y 376.037,Z 298.266,A -85,B 0,C 180,E1 -12437.608,E2 -12437.608} C_VEL
LIN {X 0,Y 375.971,Z 298.276,A -85,B 0,C 180,E1 -12440.833,E2 -12440.833} C_VEL
LIN {X 0,Y 375.987,Z 298.277,A -85,B 0,C 180,E1 -12444.282,E2 -12444.282} C_VEL
LIN {X 0,Y 376.013,Z 298.27,A -85,B 0,C 180,E1 -12446.653,E2 -12446.653} C_VEL
LIN {X 0,Y 375.958,Z 298.277,A -85,B 0,C 180,E1 -12450.313,E2 -12450.313} C_VEL
LIN {X 0,Y 375.954,Z 298.277,A -85,B 0,C 180,E1 -12454.112,E2 -12454.112} C_VEL
LIN {X 0,Y 375.948,Z 298.281,A -85,B 0,C 180,E1 -12456.742,E2 -12456.742} C_VEL
LIN {X 0,Y 375.984,Z 298.279,A -85,B 0,C 180,E1 -12459.972,E2 -12459.972} C_VEL
LIN {X 0,Y 375.929,Z 298.282,A -85,B 0,C 180,E1 -12463.766,E2 -12463.766} C_VEL
LIN {X 0,Y 376.279,Z 301.102,A -85,B 0,C 180,E1 -12466.755,E2 -12466.755} C_VEL
LIN {X 0,Y 376.387,Z 303.654,A -85,B 0,C 180,E1 -12469.193,E2 -12469.193} C_VEL
LIN {X 0,Y 376.196,Z 306.658,A -85,B 0,C 180,E1 -12471.94,E2 -12471.94} C_VEL
LIN {X 0,Y 375.97,Z 310.549,A -85,B 0,C 180,E1 -12475.335,E2 -12475.335} C_VEL
LIN {X 0,Y 375.614,Z 315.431,A -85,B 0,C 180,E1 -12479.395,E2 -12479.395} C_VEL
LIN {X 0,Y 375.345,Z 319.363,A -85,B 0,C 180,E1 -12482.551,E2 -12482.551} C_VEL
LIN {X 0,Y 376.278,Z 322.449,A -85,B 0,C 180,E1 -12482.705,E2 -12482.705} C_VEL
LIN {X 0,Y 381.387,Z 337.174,A -85,B 0,C 180,E1 -12483.55,E2 -12483.55} C_VEL
LIN {X 0,Y 385.19,Z 351.06,A -85,B 0,C 180,E1 -12484.451,E2 -12484.451} C_VEL
LIN {X 0,Y 387.522,Z 361.587,A -85,B 0,C 180,E1 -12485.227,E2 -12485.227} C_VEL
LIN {X 0,Y 386.227,Z 376.052,A -85,B 0,C 180,E1 -12486.178,E2 -12486.178} C_VEL
LIN {X 0,Y 384.631,Z 389.677,A -85,B 0,C 180,E1 -12487.295,E2 -12487.295} C_VEL
LIN {X 0,Y 382.994,Z 402.656,A -85,B 0,C 180,E1 -12488.611,E2 -12488.611} C_VEL
LIN {X 0,Y 381.566,Z 413.579,A -85,B 0,C 180,E1 -12489.945,E2 -12489.945} C_VEL
LIN {X 0,Y 380.12,Z 423.712,A -85,B 0,C 180,E1 -12491.402,E2 -12491.402} C_VEL
LIN {X 0,Y 378.561,Z 434.549,A -85,B 0,C 180,E1 -12493.277,E2 -12493.277} C_VEL
LIN {X 0,Y 377.291,Z 443.663,A -85,B 0,C 180,E1 -12495.188,E2 -12495.188} C_VEL
LIN {X 0,Y 376.444,Z 451.002,A -85,B 0,C 180,E1 -12497.055,E2 -12497.055} C_VEL
LIN {X 0,Y 375.491,Z 457.975,A -85,B 0,C 180,E1 -12499.213,E2 -12499.213} C_VEL
LIN {X 0,Y 375.004,Z 463.455,A -85,B 0,C 180,E1 -12501.378,E2 -12501.378} C_VEL
LIN {X 0,Y 374.688,Z 467.995,A -85,B 0,C 180,E1 -12503.784,E2 -12503.784} C_VEL
LIN {X 0,Y 374.547,Z 470.501,A -85,B 0,C 180,E1 -12505.696,E2 -12505.696} C_VEL
LIN {X 0,Y 374.452,Z 472.251,A -85,B 0,C 180,E1 -12507.849,E2 -12507.849} C_VEL
LIN {X 0,Y 374.472,Z 472.862,A -85,B 0,C 180,E1 -12510,E2 -12510} C_VEL
LIN {X 0,Y 374.453,Z 472.296,A -85,B 0,C 180,E1 -12512.152,E2 -12512.152} C_VEL
LIN {X 0,Y 374.546,Z 470.607,A -85,B 0,C 180,E1 -12514.305,E2 -12514.305} C_VEL
LIN {X 0,Y 374.678,Z 467.755,A -85,B 0,C 180,E1 -12516.462,E2 -12516.462} C_VEL
LIN {X 0,Y 374.998,Z 463.673,A -85,B 0,C 180,E1 -12518.623,E2 -12518.623} C_VEL
LIN {X 0,Y 375.471,Z 458.262,A -85,B 0,C 180,E1 -12520.788,E2 -12520.788} C_VEL
LIN {X 0,Y 376.401,Z 451.367,A -85,B 0,C 180,E1 -12522.948,E2 -12522.948} C_VEL
LIN {X 0,Y 377.228,Z 443.958,A -85,B 0,C 180,E1 -12524.843,E2 -12524.843} C_VEL
LIN {X 0,Y 378.505,Z 435.027,A -85,B 0,C 180,E1 -12526.726,E2 -12526.726} C_VEL
LIN {X 0,Y 379.783,Z 425.925,A -85,B 0,C 180,E1 -12528.336,E2 -12528.336} C_VEL
LIN {X 0,Y 381.364,Z 414.923,A -85,B 0,C 180,E1 -12529.972,E2 -12529.972} C_VEL
LIN {X 0,Y 383.043,Z 402.298,A -85,B 0,C 180,E1 -12531.528,E2 -12531.528} C_VEL
LIN {X 0,Y 384.688,Z 389.25,A -85,B 0,C 180,E1 -12532.844,E2 -12532.844} C_VEL
LIN {X 0,Y 386.19,Z 377.084,A -85,B 0,C 180,E1 -12533.843,E2 -12533.843} C_VEL
LIN {X 0,Y 386.838,Z 370.869,A -85,B 0,C 180,E1 -12534.285,E2 -12534.285} C_VEL
LIN {X 0,Y 386.711,Z 367.363,A -85,B 0,C 180,E1 -12534.546,E2 -12534.546} C_VEL
LIN {X 0,Y 385.863,Z 364.034,A -85,B 0,C 180,E1 -12534.832,E2 -12534.832} C_VEL
LIN {X 0,Y 382.922,Z 357.821,A -85,B 0,C 180,E1 -12535.434,E2 -12535.434} C_VEL
LIN {X 0,Y 379.392,Z 351.651,A -85,B 0,C 180,E1 -12536.04,E2 -12536.04} C_VEL
LIN {X 0,Y 377.203,Z 346.677,A -85,B 0,C 180,E1 -12536.455,E2 -12536.455} C_VEL
LIN {X 0,Y 376.694,Z 344.899,A -85,B 0,C 180,E1 -12536.58,E2 -12536.58} C_VEL
LIN {X 0,Y 372.438,Z 331.255,A -85,B 0,C 180,E1 -12537.455,E2 -12537.455} C_VEL
LIN {X 0,Y 368.422,Z 320.013,A -85,B 0,C 180,E1 -12538.096,E2 -12538.096} C_VEL
LIN {X 0,Y 368.348,Z 319.449,A -85,B 0,C 180,E1 -12538.127,E2 -12538.127} C_VEL
LIN {X 0,Y 368.593,Z 315.984,A -85,B 0,C 180,E1 -12540.985,E2 -12540.985} C_VEL
LIN {X 0,Y 368.948,Z 311.453,A -85,B 0,C 180,E1 -12544.852,E2 -12544.852} C_VEL
LIN {X 0,Y 369.26,Z 306.873,A -85,B 0,C 180,E1 -12548.908,E2 -12548.908} C_VEL
LIN {X 0,Y 369.38,Z 303.52,A -85,B 0,C 180,E1 -12552.095,E2 -12552.095} C_VEL
LIN {X 0,Y 369.083,Z 300.407,A -85,B 0,C 180,E1 -12555.207,E2 -12555.207} C_VEL
LIN {X 0,Y 368.89,Z 299.163,A -85,B 0,C 180,E1 -12556.696,E2 -12556.696} C_VEL
LIN {X 0,Y 368.911,Z 299.156,A -85,B 0,C 180,E1 -12559.643,E2 -12559.643} C_VEL
LIN {X 0,Y 368.9,Z 299.162,A -85,B 0,C 180,E1 -12563.144,E2 -12563.144} C_VEL
LIN {X 0,Y 368.895,Z 299.162,A -85,B 0,C 180,E1 -12566.462,E2 -12566.462} C_VEL
LIN {X 0,Y 368.928,Z 299.157,A -85,B 0,C 180,E1 -12569.046,E2 -12569.046} C_VEL
LIN {X 0,Y 368.873,Z 299.161,A -85,B 0,C 180,E1 -12572.789,E2 -12572.789} C_VEL
LIN {X 0,Y 368.926,Z 299.155,A -85,B 0,C 180,E1 -12576.119,E2 -12576.119} C_VEL
LIN {X 0,Y 368.935,Z 299.156,A -85,B 0,C 180,E1 -12579.947,E2 -12579.947} C_VEL
LIN {X 0,Y 368.973,Z 299.147,A -85,B 0,C 180,E1 -12583.398,E2 -12583.398} C_VEL
LIN {X 0,Y 369.055,Z 299.135,A -85,B 0,C 180,E1 -12586.79,E2 -12586.79} C_VEL
LIN {X 0,Y 369.061,Z 299.138,A -85,B 0,C 180,E1 -12590.131,E2 -12590.131} C_VEL
LIN {X 0,Y 369.159,Z 299.126,A -85,B 0,C 180,E1 -12593.441,E2 -12593.441} C_VEL
LIN {X 0,Y 369.316,Z 299.106,A -85,B 0,C 180,E1 -12597.819,E2 -12597.819} C_VEL
LIN {X 0,Y 369.428,Z 299.094,A -85,B 0,C 180,E1 -12600,E2 -12600} C_VEL
LIN {X 0,Y 369.316,Z 299.107,A -85,B 0,C 180,E1 -12602.181,E2 -12602.181} C_VEL
LIN {X 0,Y 369.159,Z 299.126,A -85,B 0,C 180,E1 -12606.559,E2 -12606.559} C_VEL
LIN {X 0,Y 369.061,Z 299.139,A -85,B 0,C 180,E1 -12609.868,E2 -12609.868} C_VEL
LIN {X 0,Y 369.035,Z 299.144,A -85,B 0,C 180,E1 -12613.772,E2 -12613.772} C_VEL
LIN {X 0,Y 368.999,Z 299.145,A -85,B 0,C 180,E1 -12617.768,E2 -12617.768} C_VEL
LIN {X 0,Y 368.907,Z 299.159,A -85,B 0,C 180,E1 -12621.221,E2 -12621.221} C_VEL
LIN {X 0,Y 368.953,Z 299.153,A -85,B 0,C 180,E1 -12624.776,E2 -12624.776} C_VEL
LIN {X 0,Y 368.961,Z 299.153,A -85,B 0,C 180,E1 -12627.204,E2 -12627.204} C_VEL
LIN {X 0,Y 368.927,Z 299.161,A -85,B 0,C 180,E1 -12630.954,E2 -12630.954} C_VEL
LIN {X 0,Y 368.927,Z 299.164,A -85,B 0,C 180,E1 -12635.001,E2 -12635.001} C_VEL
LIN {X 0,Y 368.902,Z 299.164,A -85,B 0,C 180,E1 -12638.639,E2 -12638.639} C_VEL
LIN {X 0,Y 368.907,Z 299.161,A -85,B 0,C 180,E1 -12640.371,E2 -12640.371} C_VEL
LIN {X 0,Y 369.055,Z 300.304,A -85,B 0,C 180,E1 -12642.04,E2 -12642.04} C_VEL
LIN {X 0,Y 369.636,Z 303.781,A -85,B 0,C 180,E1 -12645.293,E2 -12645.293} C_VEL
LIN {X 0,Y 369.863,Z 307.257,A -85,B 0,C 180,E1 -12648.314,E2 -12648.314} C_VEL
LIN {X 0,Y 369.687,Z 310.834,A -85,B 0,C 180,E1 -12651.209,E2 -12651.209} C_VEL
LIN {X 0,Y 369.231,Z 315.678,A -85,B 0,C 180,E1 -12654.932,E2 -12654.932} C_VEL
LIN {X 0,Y 368.895,Z 319.507,A -85,B 0,C 180,E1 -12657.762,E2 -12657.762} C_VEL
LIN {X 0,Y 368.495,Z 324.765,A -85,B 0,C 180,E1 -12661.523,E2 -12661.523} C_VEL
LIN {X 0,Y 368.476,Z 325.341,A -85,B 0,C 180,E1 -12661.928,E2 -12661.928} C_VEL
LIN {X 0,Y 369.328,Z 328.402,A -85,B 0,C 180,E1 -12662.075,E2 -12662.075} C_VEL
LIN {X 0,Y 374.147,Z 342.973,A -85,B 0,C 180,E1 -12662.908,E2 -12662.908} C_VEL
LIN {X 0,Y 377.672,Z 356.225,A -85,B 0,C 180,E1 -12663.771,E2 -12663.771} C_VEL
LIN {X 0,Y 380.559,Z 370.287,A -85,B 0,C 180,E1 -12664.811,E2 -12664.811} C_VEL
LIN {X 0,Y 380.201,Z 376.937,A -85,B 0,C 180,E1 -12665.256,E2 -12665.256} C_VEL
LIN {X 0,Y 378.718,Z 389.525,A -85,B 0,C 180,E1 -12666.195,E2 -12666.195} C_VEL
LIN {X 0,Y 377.037,Z 402.523,A -85,B 0,C 180,E1 -12667.39,E2 -12667.39} C_VEL
LIN {X 0,Y 375.249,Z 415.595,A -85,B 0,C 180,E1 -12668.867,E2 -12668.867} C_VEL
LIN {X 0,Y 373.745,Z 425.638,A -85,B 0,C 180,E1 -12670.216,E2 -12670.216} C_VEL
LIN {X 0,Y 372.25,Z 435.863,A -85,B 0,C 180,E1 -12671.849,E2 -12671.849} C_VEL
LIN {X 0,Y 370.826,Z 445.856,A -85,B 0,C 180,E1 -12673.767,E2 -12673.767} C_VEL
LIN {X 0,Y 369.625,Z 454.152,A -85,B 0,C 180,E1 -12675.689,E2 -12675.689} C_VEL
LIN {X 0,Y 368.748,Z 461.947,A -85,B 0,C 180,E1 -12677.898,E2 -12677.898} C_VEL
LIN {X 0,Y 368.026,Z 468.146,A -85,B 0,C 180,E1 -12680.103,E2 -12680.103} C_VEL
LIN {X 0,Y 367.651,Z 472.94,A -85,B 0,C 180,E1 -12682.31,E2 -12682.31} C_VEL
LIN {X 0,Y 367.428,Z 476.452,A -85,B 0,C 180,E1 -12684.512,E2 -12684.512} C_VEL
LIN {X 0,Y 367.338,Z 478.762,A -85,B 0,C 180,E1 -12686.709,E2 -12686.709} C_VEL
LIN {X 0,Y 367.347,Z 479.923,A -85,B 0,C 180,E1 -12688.903,E2 -12688.903} C_VEL
LIN {X 0,Y 367.347,Z 479.921,A -85,B 0,C 180,E1 -12691.096,E2 -12691.096} C_VEL
LIN {X 0,Y 367.339,Z 478.752,A -85,B 0,C 180,E1 -12693.29,E2 -12693.29} C_VEL
LIN {X 0,Y 367.442,Z 476.437,A -85,B 0,C 180,E1 -12695.487,E2 -12695.487} C_VEL
LIN {X 0,Y 367.668,Z 472.926,A -85,B 0,C 180,E1 -12697.689,E2 -12697.689} C_VEL
LIN {X 0,Y 368.025,Z 468.129,A -85,B 0,C 180,E1 -12699.896,E2 -12699.896} C_VEL
LIN {X 0,Y 368.741,Z 461.916,A -85,B 0,C 180,E1 -12702.101,E2 -12702.101} C_VEL
LIN {X 0,Y 369.628,Z 454.112,A -85,B 0,C 180,E1 -12704.31,E2 -12704.31} C_VEL
LIN {X 0,Y 370.82,Z 445.812,A -85,B 0,C 180,E1 -12706.233,E2 -12706.233} C_VEL
LIN {X 0,Y 372.261,Z 435.81,A -85,B 0,C 180,E1 -12708.149,E2 -12708.149} C_VEL
LIN {X 0,Y 373.808,Z 425.58,A -85,B 0,C 180,E1 -12709.78,E2 -12709.78} C_VEL
LIN {X 0,Y 375.524,Z 413.386,A -85,B 0,C 180,E1 -12711.403,E2 -12711.403} C_VEL
LIN {X 0,Y 377.381,Z 399.809,A -85,B 0,C 180,E1 -12712.876,E2 -12712.876} C_VEL
LIN {X 0,Y 379.124,Z 386.193,A -85,B 0,C 180,E1 -12714.067,E2 -12714.067} C_VEL
LIN {X 0,Y 380.614,Z 372.29,A -85,B 0,C 180,E1 -12715.043,E2 -12715.043} C_VEL
LIN {X 0,Y 380.275,Z 368.696,A -85,B 0,C 180,E1 -12715.301,E2 -12715.301} C_VEL
LIN {X 0,Y 377,Z 353.569,A -85,B 0,C 180,E1 -12716.397,E2 -12716.397} C_VEL
LIN {X 0,Y 373.006,Z 339.394,A -85,B 0,C 180,E1 -12717.295,E2 -12717.295} C_VEL
LIN {X 0,Y 368.522,Z 325.924,A -85,B 0,C 180,E1 -12718.037,E2 -12718.037} C_VEL
LIN {X 0,Y 368.461,Z 325.331,A -85,B 0,C 180,E1 -12718.08,E2 -12718.08} C_VEL
LIN {X 0,Y 368.77,Z 321.28,A -85,B 0,C 180,E1 -12720.967,E2 -12720.967} C_VEL
LIN {X 0,Y 369.227,Z 316.047,A -85,B 0,C 180,E1 -12724.821,E2 -12724.821} C_VEL
LIN {X 0,Y 369.497,Z 312.561,A -85,B 0,C 180,E1 -12727.491,E2 -12727.491} C_VEL
LIN {X 0,Y 369.823,Z 308.707,A -85,B 0,C 180,E1 -12730.523,E2 -12730.523} C_VEL
LIN {X 0,Y 369.812,Z 305.535,A -85,B 0,C 180,E1 -12733.168,E2 -12733.168} C_VEL
LIN {X 0,Y 369.382,Z 302.033,A -85,B 0,C 180,E1 -12736.301,E2 -12736.301} C_VEL
LIN {X 0,Y 369.008,Z 300.038,A -85,B 0,C 180,E1 -12738.195,E2 -12738.195} C_VEL
LIN {X 0,Y 368.906,Z 299.16,A -85,B 0,C 180,E1 -12739.642,E2 -12739.642} C_VEL
LIN {X 0,Y 368.895,Z 299.163,A -85,B 0,C 180,E1 -12743.144,E2 -12743.144} C_VEL
LIN {X 0,Y 368.89,Z 299.167,A -85,B 0,C 180,E1 -12746.461,E2 -12746.461} C_VEL
LIN {X 0,Y 368.923,Z 299.162,A -85,B 0,C 180,E1 -12749.046,E2 -12749.046} C_VEL
LIN {X 0,Y 368.956,Z 299.154,A -85,B 0,C 180,E1 -12752.796,E2 -12752.796} C_VEL
LIN {X 0,Y 368.938,Z 299.153,A -85,B 0,C 180,E1 -12756.113,E2 -12756.113} C_VEL
LIN {X 0,Y 368.929,Z 299.156,A -85,B 0,C 180,E1 -12759.947,E2 -12759.947} C_VEL
LIN {X 0,Y 368.968,Z 299.152,A -85,B 0,C 180,E1 -12763.398,E2 -12763.398} C_VEL
LIN {X 0,Y 369.05,Z 299.139,A -85,B 0,C 180,E1 -12766.79,E2 -12766.79} C_VEL
LIN {X 0,Y 369.056,Z 299.138,A -85,B 0,C 180,E1 -12770.132,E2 -12770.132} C_VEL
LIN {X 0,Y 369.154,Z 299.127,A -85,B 0,C 180,E1 -12773.441,E2 -12773.441} C_VEL
LIN {X 0,Y 369.311,Z 299.102,A -85,B 0,C 180,E1 -12777.819,E2 -12777.819} C_VEL
LIN {X 0,Y 369.446,Z 299.092,A -85,B 0,C 180,E1 -12780,E2 -12780} C_VEL
LIN {X 0,Y 369.311,Z 299.106,A -85,B 0,C 180,E1 -12782.181,E2 -12782.181} C_VEL
LIN {X 0,Y 369.154,Z 299.127,A -85,B 0,C 180,E1 -12786.559,E2 -12786.559} C_VEL
LIN {X 0,Y 369.056,Z 299.139,A -85,B 0,C 180,E1 -12789.869,E2 -12789.869} C_VEL
LIN {X 0,Y 369.03,Z 299.143,A -85,B 0,C 180,E1 -12793.773,E2 -12793.773} C_VEL
LIN {X 0,Y 368.994,Z 299.144,A -85,B 0,C 180,E1 -12797.769,E2 -12797.769} C_VEL
LIN {X 0,Y 368.923,Z 299.156,A -85,B 0,C 180,E1 -12801.22,E2 -12801.22} C_VEL
LIN {X 0,Y 368.951,Z 299.152,A -85,B 0,C 180,E1 -12804.776,E2 -12804.776} C_VEL
LIN {X 0,Y 368.957,Z 299.15,A -85,B 0,C 180,E1 -12807.204,E2 -12807.204} C_VEL
LIN {X 0,Y 368.923,Z 299.153,A -85,B 0,C 180,E1 -12810.954,E2 -12810.954} C_VEL
LIN {X 0,Y 368.923,Z 299.154,A -85,B 0,C 180,E1 -12815.002,E2 -12815.002} C_VEL
LIN {X 0,Y 368.904,Z 299.159,A -85,B 0,C 180,E1 -12818.641,E2 -12818.641} C_VEL
LIN {X 0,Y 368.877,Z 299.164,A -85,B 0,C 180,E1 -12822.01,E2 -12822.01} C_VEL
LIN {X 0,Y 368.882,Z 299.179,A -85,B 0,C 180,E1 -12823.617,E2 -12823.617} C_VEL
LIN {X 0,Y 369.276,Z 302.191,A -85,B 0,C 180,E1 -12826.754,E2 -12826.754} C_VEL
LIN {X 0,Y 369.401,Z 303.697,A -85,B 0,C 180,E1 -12828.251,E2 -12828.251} C_VEL
LIN {X 0,Y 369.238,Z 306.944,A -85,B 0,C 180,E1 -12831.296,E2 -12831.296} C_VEL
LIN {X 0,Y 368.943,Z 311.264,A -85,B 0,C 180,E1 -12835.148,E2 -12835.148} C_VEL
LIN {X 0,Y 368.585,Z 315.917,A -85,B 0,C 180,E1 -12839.097,E2 -12839.097} C_VEL
LIN {X 0,Y 368.353,Z 319.427,A -85,B 0,C 180,E1 -12841.978,E2 -12841.978} C_VEL
LIN {X 0,Y 369.315,Z 322.627,A -85,B 0,C 180,E1 -12842.148,E2 -12842.148} C_VEL
LIN {X 0,Y 374.462,Z 337.347,A -85,B 0,C 180,E1 -12843.026,E2 -12843.026} C_VEL
LIN {X 0,Y 378.201,Z 350.638,A -85,B 0,C 180,E1 -12843.917,E2 -12843.917} C_VEL
LIN {X 0,Y 380.964,Z 363.56,A -85,B 0,C 180,E1 -12844.894,E2 -12844.894} C_VEL
LIN {X 0,Y 379.581,Z 377.631,A -85,B 0,C 180,E1 -12845.858,E2 -12845.858} C_VEL
LIN {X 0,Y 377.893,Z 391.176,A -85,B 0,C 180,E1 -12847.012,E2 -12847.012} C_VEL
LIN {X 0,Y 376.193,Z 403.901,A -85,B 0,C 180,E1 -12848.349,E2 -12848.349} C_VEL
LIN {X 0,Y 374.525,Z 416.099,A -85,B 0,C 180,E1 -12849.911,E2 -12849.911} C_VEL
LIN {X 0,Y 372.839,Z 427.047,A -85,B 0,C 180,E1 -12851.595,E2 -12851.595} C_VEL
LIN {X 0,Y 371.335,Z 437.321,A -85,B 0,C 180,E1 -12853.508,E2 -12853.508} C_VEL
LIN {X 0,Y 370.072,Z 445.853,A -85,B 0,C 180,E1 -12855.427,E2 -12855.427} C_VEL
LIN {X 0,Y 369.217,Z 452.953,A -85,B 0,C 180,E1 -12857.356,E2 -12857.356} C_VEL
LIN {X 0,Y 368.336,Z 459.542,A -85,B 0,C 180,E1 -12859.557,E2 -12859.557} C_VEL
LIN {X 0,Y 367.845,Z 464.694,A -85,B 0,C 180,E1 -12861.762,E2 -12861.762} C_VEL
LIN {X 0,Y 367.612,Z 468.273,A -85,B 0,C 180,E1 -12863.792,E2 -12863.792} C_VEL
LIN {X 0,Y 367.455,Z 470.57,A -85,B 0,C 180,E1 -12865.613,E2 -12865.613} C_VEL
LIN {X 0,Y 367.353,Z 472.32,A -85,B 0,C 180,E1 -12867.808,E2 -12867.808} C_VEL
LIN {X 0,Y 367.373,Z 472.931,A -85,B 0,C 180,E1 -12870,E2 -12870} C_VEL
LIN {X 0,Y 367.354,Z 472.365,A -85,B 0,C 180,E1 -12872.193,E2 -12872.193} C_VEL
LIN {X 0,Y 367.454,Z 470.675,A -85,B 0,C 180,E1 -12874.388,E2 -12874.388} C_VEL
LIN {X 0,Y 367.592,Z 467.823,A -85,B 0,C 180,E1 -12876.587,E2 -12876.587} C_VEL
LIN {X 0,Y 367.957,Z 463.741,A -85,B 0,C 180,E1 -12878.79,E2 -12878.79} C_VEL
LIN {X 0,Y 368.457,Z 458.33,A -85,B 0,C 180,E1 -12880.996,E2 -12880.996} C_VEL
LIN {X 0,Y 369.385,Z 451.435,A -85,B 0,C 180,E1 -12883.198,E2 -12883.198} C_VEL
LIN {X 0,Y 370.306,Z 444.024,A -85,B 0,C 180,E1 -12885.127,E2 -12885.127} C_VEL
LIN {X 0,Y 371.671,Z 435.094,A -85,B 0,C 180,E1 -12887.043,E2 -12887.043} C_VEL
LIN {X 0,Y 373.037,Z 425.991,A -85,B 0,C 180,E1 -12888.68,E2 -12888.68} C_VEL
LIN {X 0,Y 374.721,Z 414.673,A -85,B 0,C 180,E1 -12890.388,E2 -12890.388} C_VEL
LIN {X 0,Y 376.446,Z 402.363,A -85,B 0,C 180,E1 -12891.925,E2 -12891.925} C_VEL
LIN {X 0,Y 378.127,Z 389.314,A -85,B 0,C 180,E1 -12893.264,E2 -12893.264} C_VEL
LIN {X 0,Y 379.857,Z 375.998,A -85,B 0,C 180,E1 -12894.36,E2 -12894.36} C_VEL
LIN {X 0,Y 381.045,Z 363.454,A -85,B 0,C 180,E1 -12895.208,E2 -12895.208} C_VEL
LIN {X 0,Y 377.887,Z 349.363,A -85,B 0,C 180,E1 -12896.271,E2 -12896.271} C_VEL
LIN {X 0,Y 376.694,Z 344.899,A -85,B 0,C 180,E1 -12896.58,E2 -12896.58} C_VEL
LIN {X 0,Y 375.152,Z 341.687,A -85,B 0,C 180,E1 -12896.852,E2 -12896.852} C_VEL
LIN {X 0,Y 370.925,Z 337.527,A -85,B 0,C 180,E1 -12897.361,E2 -12897.361} C_VEL
LIN {X 0,Y 366.657,Z 333.322,A -85,B 0,C 180,E1 -12897.857,E2 -12897.857} C_VEL
LIN {X 0,Y 365.041,Z 330.042,A -85,B 0,C 180,E1 -12898.104,E2 -12898.104} C_VEL
LIN {X 0,Y 361.427,Z 320.181,A -85,B 0,C 180,E1 -12898.687,E2 -12898.687} C_VEL
LIN {X 0,Y 361.319,Z 319.481,A -85,B 0,C 180,E1 -12898.756,E2 -12898.756} C_VEL
LIN {X 0,Y 361.562,Z 316.063,A -85,B 0,C 180,E1 -12901.656,E2 -12901.656} C_VEL
LIN {X 0,Y 361.944,Z 311.79,A -85,B 0,C 180,E1 -12905.36,E2 -12905.36} C_VEL
LIN {X 0,Y 362.234,Z 307.704,A -85,B 0,C 180,E1 -12909.097,E2 -12909.097} C_VEL
LIN {X 0,Y 362.348,Z 305.45,A -85,B 0,C 180,E1 -12911.258,E2 -12911.258} C_VEL
LIN {X 0,Y 362.188,Z 302.582,A -85,B 0,C 180,E1 -12914.114,E2 -12914.114} C_VEL
LIN {X 0,Y 361.958,Z 300.87,A -85,B 0,C 180,E1 -12915.923,E2 -12915.923} C_VEL
LIN {X 0,Y 361.837,Z 300.041,A -85,B 0,C 180,E1 -12917.568,E2 -12917.568} C_VEL
LIN {X 0,Y 361.869,Z 300.035,A -85,B 0,C 180,E1 -12920.973,E2 -12920.973} C_VEL
LIN {X 0,Y 361.873,Z 300.037,A -85,B 0,C 180,E1 -12924.655,E2 -12924.655} C_VEL
LIN {X 0,Y 361.836,Z 300.04,A -85,B 0,C 180,E1 -12928.37,E2 -12928.37} C_VEL
LIN {X 0,Y 361.864,Z 300.036,A -85,B 0,C 180,E1 -12930.952,E2 -12930.952} C_VEL
LIN {X 0,Y 361.888,Z 300.032,A -85,B 0,C 180,E1 -12934.707,E2 -12934.707} C_VEL
LIN {X 0,Y 361.859,Z 300.034,A -85,B 0,C 180,E1 -12938.345,E2 -12938.345} C_VEL
LIN {X 0,Y 361.966,Z 300.023,A -85,B 0,C 180,E1 -12942.061,E2 -12942.061} C_VEL
LIN {X 0,Y 361.996,Z 300.02,A -85,B 0,C 180,E1 -12946.101,E2 -12946.101} C_VEL
LIN {X 0,Y 361.998,Z 300.018,A -85,B 0,C 180,E1 -12949.937,E2 -12949.937} C_VEL
LIN {X 0,Y 362.122,Z 300.002,A -85,B 0,C 180,E1 -12953.313,E2 -12953.313} C_VEL
LIN {X 0,Y 362.28,Z 299.982,A -85,B 0,C 180,E1 -12957.776,E2 -12957.776} C_VEL
LIN {X 0,Y 362.379,Z 299.972,A -85,B 0,C 180,E1 -12960,E2 -12960} C_VEL
LIN {X 0,Y 362.28,Z 299.983,A -85,B 0,C 180,E1 -12962.223,E2 -12962.223} C_VEL
LIN {X 0,Y 362.122,Z 300.002,A -85,B 0,C 180,E1 -12966.687,E2 -12966.687} C_VEL
LIN {X 0,Y 361.998,Z 300.018,A -85,B 0,C 180,E1 -12970.063,E2 -12970.063} C_VEL
LIN {X 0,Y 361.995,Z 300.02,A -85,B 0,C 180,E1 -12973.899,E2 -12973.899} C_VEL
LIN {X 0,Y 361.965,Z 300.022,A -85,B 0,C 180,E1 -12977.939,E2 -12977.939} C_VEL
LIN {X 0,Y 361.859,Z 300.037,A -85,B 0,C 180,E1 -12981.655,E2 -12981.655} C_VEL
LIN {X 0,Y 361.925,Z 300.026,A -85,B 0,C 180,E1 -12985.29,E2 -12985.29} C_VEL
LIN {X 0,Y 361.906,Z 300.033,A -85,B 0,C 180,E1 -12987.779,E2 -12987.779} C_VEL
LIN {X 0,Y 361.835,Z 300.044,A -85,B 0,C 180,E1 -12991.629,E2 -12991.629} C_VEL
LIN {X 0,Y 361.872,Z 300.043,A -85,B 0,C 180,E1 -12995.345,E2 -12995.345} C_VEL
LIN {X 0,Y 361.864,Z 300.04,A -85,B 0,C 180,E1 -12999.026,E2 -12999.026} C_VEL
LIN {X 0,Y 361.864,Z 300.259,A -85,B 0,C 180,E1 -13000.761,E2 -13000.761} C_VEL
LIN {X 0,Y 362.48,Z 303.837,A -85,B 0,C 180,E1 -13004.266,E2 -13004.266} C_VEL
LIN {X 0,Y 362.828,Z 307.305,A -85,B 0,C 180,E1 -13007.397,E2 -13007.397} C_VEL
LIN {X 0,Y 362.719,Z 310.699,A -85,B 0,C 180,E1 -13010.253,E2 -13010.253} C_VEL
LIN {X 0,Y 362.421,Z 314.192,A -85,B 0,C 180,E1 -13013.048,E2 -13013.048} C_VEL
LIN {X 0,Y 361.985,Z 318.819,A -85,B 0,C 180,E1 -13016.6,E2 -13016.6} C_VEL
LIN {X 0,Y 361.606,Z 322.942,A -85,B 0,C 180,E1 -13019.647,E2 -13019.647} C_VEL
LIN {X 0,Y 361.446,Z 325.26,A -85,B 0,C 180,E1 -13021.328,E2 -13021.328} C_VEL
LIN {X 0,Y 363.349,Z 331.171,A -85,B 0,C 180,E1 -13021.648,E2 -13021.648} C_VEL
LIN {X 0,Y 368.05,Z 345.753,A -85,B 0,C 180,E1 -13022.541,E2 -13022.541} C_VEL
LIN {X 0,Y 371.269,Z 358.049,A -85,B 0,C 180,E1 -13023.383,E2 -13023.383} C_VEL
LIN {X 0,Y 373.991,Z 371.535,A -85,B 0,C 180,E1 -13024.423,E2 -13024.423} C_VEL
LIN {X 0,Y 373.849,Z 375.822,A -85,B 0,C 180,E1 -13024.728,E2 -13024.728} C_VEL
LIN {X 0,Y 372.195,Z 389.46,A -85,B 0,C 180,E1 -13025.751,E2 -13025.751} C_VEL
LIN {X 0,Y 370.469,Z 402.457,A -85,B 0,C 180,E1 -13026.967,E2 -13026.967} C_VEL
LIN {X 0,Y 368.581,Z 415.528,A -85,B 0,C 180,E1 -13028.466,E2 -13028.466} C_VEL
LIN {X 0,Y 366.762,Z 427.407,A -85,B 0,C 180,E1 -13030.123,E2 -13030.123} C_VEL
LIN {X 0,Y 365.218,Z 437.308,A -85,B 0,C 180,E1 -13031.778,E2 -13031.778} C_VEL
LIN {X 0,Y 363.751,Z 447.043,A -85,B 0,C 180,E1 -13033.73,E2 -13033.73} C_VEL
LIN {X 0,Y 362.403,Z 455.729,A -85,B 0,C 180,E1 -13035.845,E2 -13035.845} C_VEL
LIN {X 0,Y 361.756,Z 461.879,A -85,B 0,C 180,E1 -13037.66,E2 -13037.66} C_VEL
LIN {X 0,Y 360.976,Z 468.077,A -85,B 0,C 180,E1 -13039.908,E2 -13039.908} C_VEL
LIN {X 0,Y 360.583,Z 472.872,A -85,B 0,C 180,E1 -13042.158,E2 -13042.158} C_VEL
LIN {X 0,Y 360.337,Z 476.383,A -85,B 0,C 180,E1 -13044.403,E2 -13044.403} C_VEL
LIN {X 0,Y 360.259,Z 478.693,A -85,B 0,C 180,E1 -13046.644,E2 -13046.644} C_VEL
LIN {X 0,Y 360.245,Z 479.854,A -85,B 0,C 180,E1 -13048.882,E2 -13048.882} C_VEL
LIN {X 0,Y 360.245,Z 479.852,A -85,B 0,C 180,E1 -13051.117,E2 -13051.117} C_VEL
LIN {X 0,Y 360.26,Z 478.683,A -85,B 0,C 180,E1 -13053.355,E2 -13053.355} C_VEL
LIN {X 0,Y 360.35,Z 476.367,A -85,B 0,C 180,E1 -13055.596,E2 -13055.596} C_VEL
LIN {X 0,Y 360.594,Z 472.856,A -85,B 0,C 180,E1 -13057.841,E2 -13057.841} C_VEL
LIN {X 0,Y 360.975,Z 468.058,A -85,B 0,C 180,E1 -13060.091,E2 -13060.091} C_VEL
LIN {X 0,Y 361.75,Z 461.845,A -85,B 0,C 180,E1 -13062.339,E2 -13062.339} C_VEL
LIN {X 0,Y 362.693,Z 454.04,A -85,B 0,C 180,E1 -13064.59,E2 -13064.59} C_VEL
LIN {X 0,Y 363.929,Z 445.74,A -85,B 0,C 180,E1 -13066.549,E2 -13066.549} C_VEL
LIN {X 0,Y 365.472,Z 435.738,A -85,B 0,C 180,E1 -13068.499,E2 -13068.499} C_VEL
LIN {X 0,Y 367.062,Z 425.507,A -85,B 0,C 180,E1 -13070.159,E2 -13070.159} C_VEL
LIN {X 0,Y 368.888,Z 413.314,A -85,B 0,C 180,E1 -13071.808,E2 -13071.808} C_VEL
LIN {X 0,Y 370.838,Z 399.736,A -85,B 0,C 180,E1 -13073.304,E2 -13073.304} C_VEL
LIN {X 0,Y 372.642,Z 386.119,A -85,B 0,C 180,E1 -13074.513,E2 -13074.513} C_VEL
LIN {X 0,Y 374.114,Z 372.781,A -85,B 0,C 180,E1 -13075.468,E2 -13075.468} C_VEL
LIN {X 0,Y 371.61,Z 359.99,A -85,B 0,C 180,E1 -13076.466,E2 -13076.466} C_VEL
LIN {X 0,Y 368.391,Z 347.02,A -85,B 0,C 180,E1 -13077.365,E2 -13077.365} C_VEL
LIN {X 0,Y 363.644,Z 331.867,A -85,B 0,C 180,E1 -13078.293,E2 -13078.293} C_VEL
LIN {X 0,Y 361.504,Z 325.799,A -85,B 0,C 180,E1 -13078.631,E2 -13078.631} C_VEL
LIN {X 0,Y 361.446,Z 325.224,A -85,B 0,C 180,E1 -13078.698,E2 -13078.698} C_VEL
LIN {X 0,Y 361.78,Z 321.205,A -85,B 0,C 180,E1 -13081.634,E2 -13081.634} C_VEL
LIN {X 0,Y 362.217,Z 316.207,A -85,B 0,C 180,E1 -13085.421,E2 -13085.421} C_VEL
LIN {X 0,Y 362.589,Z 312.497,A -85,B 0,C 180,E1 -13088.333,E2 -13088.333} C_VEL
LIN {X 0,Y 362.811,Z 308.982,A -85,B 0,C 180,E1 -13091.193,E2 -13091.193} C_VEL
LIN {X 0,Y 362.693,Z 305.478,A -85,B 0,C 180,E1 -13094.232,E2 -13094.232} C_VEL
LIN {X 0,Y 362.136,Z 301.974,A -85,B 0,C 180,E1 -13097.515,E2 -13097.515} C_VEL
LIN {X 0,Y 361.859,Z 300.226,A -85,B 0,C 180,E1 -13099.239,E2 -13099.239} C_VEL
LIN {X 0,Y 361.862,Z 300.038,A -85,B 0,C 180,E1 -13101.575,E2 -13101.575} C_VEL
LIN {X 0,Y 361.868,Z 300.04,A -85,B 0,C 180,E1 -13104.655,E2 -13104.655} C_VEL
LIN {X 0,Y 361.831,Z 300.045,A -85,B 0,C 180,E1 -13108.37,E2 -13108.37} C_VEL
LIN {X 0,Y 361.901,Z 300.036,A -85,B 0,C 180,E1 -13112.221,E2 -13112.221} C_VEL
LIN {X 0,Y 361.921,Z 300.028,A -85,B 0,C 180,E1 -13114.71,E2 -13114.71} C_VEL
LIN {X 0,Y 361.885,Z 300.033,A -85,B 0,C 180,E1 -13118.347,E2 -13118.347} C_VEL
LIN {X 0,Y 361.96,Z 300.022,A -85,B 0,C 180,E1 -13122.061,E2 -13122.061} C_VEL
LIN {X 0,Y 361.99,Z 300.019,A -85,B 0,C 180,E1 -13126.101,E2 -13126.101} C_VEL
LIN {X 0,Y 361.993,Z 300.018,A -85,B 0,C 180,E1 -13129.937,E2 -13129.937} C_VEL
LIN {X 0,Y 362.117,Z 300.003,A -85,B 0,C 180,E1 -13133.313,E2 -13133.313} C_VEL
LIN {X 0,Y 362.275,Z 299.978,A -85,B 0,C 180,E1 -13137.777,E2 -13137.777} C_VEL
LIN {X 0,Y 362.395,Z 299.97,A -85,B 0,C 180,E1 -13140,E2 -13140} C_VEL
LIN {X 0,Y 362.275,Z 299.982,A -85,B 0,C 180,E1 -13142.224,E2 -13142.224} C_VEL
LIN {X 0,Y 362.117,Z 300.003,A -85,B 0,C 180,E1 -13146.687,E2 -13146.687} C_VEL
LIN {X 0,Y 361.993,Z 300.019,A -85,B 0,C 180,E1 -13150.063,E2 -13150.063} C_VEL
LIN {X 0,Y 361.991,Z 300.019,A -85,B 0,C 180,E1 -13153.899,E2 -13153.899} C_VEL
LIN {X 0,Y 361.96,Z 300.02,A -85,B 0,C 180,E1 -13157.939,E2 -13157.939} C_VEL
LIN {X 0,Y 361.887,Z 300.033,A -85,B 0,C 180,E1 -13161.653,E2 -13161.653} C_VEL
LIN {X 0,Y 361.922,Z 300.027,A -85,B 0,C 180,E1 -13165.291,E2 -13165.291} C_VEL
LIN {X 0,Y 361.902,Z 300.029,A -85,B 0,C 180,E1 -13167.78,E2 -13167.78} C_VEL
LIN {X 0,Y 361.832,Z 300.035,A -85,B 0,C 180,E1 -13171.63,E2 -13171.63} C_VEL
LIN {X 0,Y 361.869,Z 300.033,A -85,B 0,C 180,E1 -13175.345,E2 -13175.345} C_VEL
LIN {X 0,Y 361.865,Z 300.036,A -85,B 0,C 180,E1 -13179.027,E2 -13179.027} C_VEL
LIN {X 0,Y 361.833,Z 300.043,A -85,B 0,C 180,E1 -13182.83,E2 -13182.83} C_VEL
LIN {X 0,Y 361.969,Z 301.003,A -85,B 0,C 180,E1 -13184.345,E2 -13184.345} C_VEL
LIN {X 0,Y 362.329,Z 304.002,A -85,B 0,C 180,E1 -13187.483,E2 -13187.483} C_VEL
LIN {X 0,Y 362.268,Z 306.778,A -85,B 0,C 180,E1 -13190.195,E2 -13190.195} C_VEL
LIN {X 0,Y 362.04,Z 309.81,A -85,B 0,C 180,E1 -13193.004,E2 -13193.004} C_VEL
LIN {X 0,Y 361.812,Z 312.849,A -85,B 0,C 180,E1 -13195.716,E2 -13195.716} C_VEL
LIN {X 0,Y 361.462,Z 317.413,A -85,B 0,C 180,E1 -13199.635,E2 -13199.635} C_VEL
LIN {X 0,Y 361.33,Z 319.502,A -85,B 0,C 180,E1 -13201.386,E2 -13201.386} C_VEL
LIN {X 0,Y 362.279,Z 322.617,A -85,B 0,C 180,E1 -13201.556,E2 -13201.556} C_VEL
LIN {X 0,Y 367.544,Z 337.312,A -85,B 0,C 180,E1 -13202.47,E2 -13202.47} C_VEL
LIN {X 0,Y 371.247,Z 350.489,A -85,B 0,C 180,E1 -13203.378,E2 -13203.378} C_VEL
LIN {X 0,Y 374.23,Z 363.641,A -85,B 0,C 180,E1 -13204.41,E2 -13204.41} C_VEL
LIN {X 0,Y 374.273,Z 367.081,A -85,B 0,C 180,E1 -13204.654,E2 -13204.654} C_VEL
LIN {X 0,Y 372.746,Z 380.668,A -85,B 0,C 180,E1 -13205.642,E2 -13205.642} C_VEL
LIN {X 0,Y 370.993,Z 394.049,A -85,B 0,C 180,E1 -13206.854,E2 -13206.854} C_VEL
LIN {X 0,Y 369.278,Z 406.31,A -85,B 0,C 180,E1 -13208.216,E2 -13208.216} C_VEL
LIN {X 0,Y 367.46,Z 418.525,A -85,B 0,C 180,E1 -13209.864,E2 -13209.864} C_VEL
LIN {X 0,Y 365.841,Z 428.743,A -85,B 0,C 180,E1 -13211.521,E2 -13211.521} C_VEL
LIN {X 0,Y 364.278,Z 438.742,A -85,B 0,C 180,E1 -13213.468,E2 -13213.468} C_VEL
LIN {X 0,Y 362.88,Z 447.549,A -85,B 0,C 180,E1 -13215.55,E2 -13215.55} C_VEL
LIN {X 0,Y 361.99,Z 454.828,A -85,B 0,C 180,E1 -13217.669,E2 -13217.669} C_VEL
LIN {X 0,Y 361.16,Z 461.033,A -85,B 0,C 180,E1 -13219.914,E2 -13219.914} C_VEL
LIN {X 0,Y 360.681,Z 465.824,A -85,B 0,C 180,E1 -13222.161,E2 -13222.161} C_VEL
LIN {X 0,Y 360.429,Z 469.335,A -85,B 0,C 180,E1 -13224.406,E2 -13224.406} C_VEL
LIN {X 0,Y 360.295,Z 471.657,A -85,B 0,C 180,E1 -13226.646,E2 -13226.646} C_VEL
LIN {X 0,Y 360.256,Z 472.842,A -85,B 0,C 180,E1 -13228.883,E2 -13228.883} C_VEL
LIN {X 0,Y 360.256,Z 472.857,A -85,B 0,C 180,E1 -13231.118,E2 -13231.118} C_VEL
LIN {X 0,Y 360.294,Z 471.731,A -85,B 0,C 180,E1 -13233.355,E2 -13233.355} C_VEL
LIN {X 0,Y 360.427,Z 469.467,A -85,B 0,C 180,E1 -13235.595,E2 -13235.595} C_VEL
LIN {X 0,Y 360.68,Z 466.009,A -85,B 0,C 180,E1 -13237.84,E2 -13237.84} C_VEL
LIN {X 0,Y 361.132,Z 461.278,A -85,B 0,C 180,E1 -13240.088,E2 -13240.088} C_VEL
LIN {X 0,Y 361.956,Z 455.147,A -85,B 0,C 180,E1 -13242.333,E2 -13242.333} C_VEL
LIN {X 0,Y 362.93,Z 447.432,A -85,B 0,C 180,E1 -13244.581,E2 -13244.581} C_VEL
LIN {X 0,Y 364.198,Z 439.206,A -85,B 0,C 180,E1 -13246.537,E2 -13246.537} C_VEL
LIN {X 0,Y 365.724,Z 429.298,A -85,B 0,C 180,E1 -13248.486,E2 -13248.486} C_VEL
LIN {X 0,Y 367.55,Z 418.068,A -85,B 0,C 180,E1 -13250.304,E2 -13250.304} C_VEL
LIN {X 0,Y 369.341,Z 405.943,A -85,B 0,C 180,E1 -13251.928,E2 -13251.928} C_VEL
LIN {X 0,Y 371.067,Z 393.632,A -85,B 0,C 180,E1 -13253.289,E2 -13253.289} C_VEL
LIN {X 0,Y 372.848,Z 380.175,A -85,B 0,C 180,E1 -13254.5,E2 -13254.5} C_VEL
LIN {X 0,Y 374.297,Z 366.962,A -85,B 0,C 180,E1 -13255.456,E2 -13255.456} C_VEL
LIN {X 0,Y 374.306,Z 363.794,A -85,B 0,C 180,E1 -13255.677,E2 -13255.677} C_VEL
LIN {X 0,Y 370.994,Z 349.333,A -85,B 0,C 180,E1 -13256.803,E2 -13256.803} C_VEL
LIN {X 0,Y 367.05,Z 335.95,A -85,B 0,C 180,E1 -13257.732,E2 -13257.732} C_VEL
LIN {X 0,Y 365.041,Z 330.042,A -85,B 0,C 180,E1 -13258.104,E2 -13258.104} C_VEL
LIN {X 0,Y 363.366,Z 326.577,A -85,B 0,C 180,E1 -13258.358,E2 -13258.358} C_VEL
LIN {X 0,Y 360.857,Z 323.822,A -85,B 0,C 180,E1 -13258.68,E2 -13258.68} C_VEL
LIN {X 0,Y 357.349,Z 321.04,A -85,B 0,C 180,E1 -13259.222,E2 -13259.222} C_VEL
LIN {X 0,Y 355.261,Z 319.495,A -85,B 0,C 180,E1 -13259.737,E2 -13259.737} C_VEL
LIN {X 0,Y 354.395,Z 318.5,A -85,B 0,C 180,E1 -13260.294,E2 -13260.294} C_VEL
LIN {X 0,Y 354.393,Z 318.435,A -85,B 0,C 180,E1 -13260.347,E2 -13260.347} C_VEL
LIN {X 0,Y 354.714,Z 314.584,A -85,B 0,C 180,E1 -13263.695,E2 -13263.695} C_VEL
LIN {X 0,Y 354.954,Z 311.559,A -85,B 0,C 180,E1 -13266.441,E2 -13266.441} C_VEL
LIN {X 0,Y 355.23,Z 308.319,A -85,B 0,C 180,E1 -13269.503,E2 -13269.503} C_VEL
LIN {X 0,Y 355.329,Z 305.489,A -85,B 0,C 180,E1 -13272.259,E2 -13272.259} C_VEL
LIN {X 0,Y 355.018,Z 302.448,A -85,B 0,C 180,E1 -13275.452,E2 -13275.452} C_VEL
LIN {X 0,Y 354.792,Z 300.922,A -85,B 0,C 180,E1 -13277.132,E2 -13277.132} C_VEL
LIN {X 0,Y 354.815,Z 300.915,A -85,B 0,C 180,E1 -13280.666,E2 -13280.666} C_VEL
